    stTargetAssertion := i_stRequestedAssertion;
    nTargetAssertionID := i_nRequestedAssertionID;
	
	LogActions('New target set');
	
    xNewBP := TRUE;
    
ELSE
    IF NOT F_ValidReqID(i_nRequestedAssertionID) THEN
        
        nErrID := PMPS_CODES.BadTargetID;
    ELSIF NOT F_ValidReqID(i_TransitionAssertionID) THEN
        nErrID := PMPS_CODES.BadTransID;
	END_IF
    LogActions('Error in set new target');
    bError := TRUE;
END_IF
END_ACTION

ACTION WaitingForFinalAssertion_DO:
//Final Assertion Verification

xFinalBPInArb := fbArbiter.CheckRequest( i_nRequestedAssertionID);;
END_ACTION

ACTION WaitingForFinalAssertion_EXIT:
//Set this bool false so we can get a rising edge on the next try
xFinalBP := FALSE;
END_ACTION

ACTION WaitingForTransitionAssertion_DO:
//Transition Assertion Verification
xTranBP    := F_SafeBPCompare0Rate(stCurrentBeamParameters, i_stTransitionAssertion) AND
    fbArbiter.CheckRequest(i_TransitionAssertionID);
END_ACTION

ACTION WaitingForTransitionAssertion_EXIT:
xTranBP := FALSE;
END_ACTION

END_FUNCTION_BLOCK

// MajorComponents/InterPlcComm/FB_ArbiterToSubSys_IO
(* Exchanges preemption requests and current beam state with subsystems in arbiter
network.

2019-12-2, A. Wallace

Use in conjunction with FB_SubSysToArbiter_IO.

This FB runs in the beamline arbiter PLC (BAP). There should be one of these for every
subsystem interfaced to the BAP. Each subsystem PLC should run a sibling FB_SubSysToArbiter_IO FB.

This FB and its subordinate communicate through the ethercat connection between the subsystem PLC and the BAP.

A beam parameter set request is sent from the subsystem to this PLC, and includes a cohort number.

This cohort number (i_RequestedBP.nCohortInt) is compared to a local cohort number (nRequestedCohort). 
A request from the subsystem to update or modify its current request is indicated by an increase in the
i_RequestedBP.nCohortInt value. Then this function block updates the local arbiter request for the subsystem
and awaits confirmation. Once the new request is confirmed in the preemptive system this function block increments
the ActiveCohort value to match the nRequestedCohort. ActiveCohort is also relayed back to the subsystem
as the active cohort value in the o_CurrentBP set. The subsystem then knows its request has been heard,
and can carry out its own acknowledgement to its various requestors.

Things to note:
If a subsystem has any new or changed preemptive requests you should see the cohort value increment a bit.
If the cohort number is incrementing out of control, it usually means the subsysetm has some preemptive
request loop (two arbiters elevating to each other), or there is a RequestAdd, RequestRemove loop.

*)
FUNCTION_BLOCK FB_ArbiterToSubSys_IO
VAR_INPUT
	RequestingSystemID	:	DWORD := PMPS_GVL.EXCLUDED_ASSERTION_ID; // System ID for making requests to the supreme arbiter
    sName : STRING := 'ArbiterToSubSys';
    Reset : BOOL;
END_VAR
VAR_OUTPUT
END_VAR
VAR_IN_OUT
	Arbiter	: FB_Arbiter;
    fbFFHWO : FB_HardwareFFOutput;
END_VAR
VAR
    
	i_RequestedBP AT %I*	:	ST_BeamParams_IO; // Requested BP from subsystem
    {attribute 'pytmc' := '
        pv: RequestedBP:FromSubSys
    '}
    RequestedBP: ST_BeamParams;
    
	o_CurrentBP AT %Q* : ST_BeamParams_IO; // Current BP set
    
    // EL6692 Diagnostics
    i_Connected AT %I* : BOOL; // SYNC Inputs^External device not connected !!! Doesn't really work.
    {attribute 'pytmc' := 'pv: WcState
        io: i
        field: DESC Working counter state.
        field: ZNAM OK
        field: ONAM Error'}
    i_WcState AT %I* : BOOL := TRUE; // WcState^WcState
    {attribute 'pytmc' := 'pv: TxPDO_state
        io: i
        field: DESC PDO Transmission is OK
        field: ZNAM OK
        field: ONAM Error'}
    i_TxPDOState AT %I* : BOOL := TRUE; // SYNC Inputs^TxPDO state
    {attribute 'pytmc' := 'pv: TxPDO_toggle
        io: i
        field: DESC PDO Transmission is OK
        field: ZNAM OK
        field: ONAM Error'}
    i_TxPDOToggle AT %I* : BOOL; // TxPDO toggle
    
    // Fast faults
    ffPMPSIO_Disconnect : FB_FastFault := (i_Desc:='Issue w/ arbiter interface to subsystem, verify subsystem is OK, or ethercat connection.'); // Fast fault for ethercat issues
    nActiveCohort : UDINT := 0; // Active cohort. Updated to the req. number from the sub system after request is confirmed.
    nRequestedCohort : UDINT := 0;
    rtToggle : R_TRIG;

	
END_VAR


// Incoming request from subsystem PLC
RequestedBP := IO_TO_BP(i_RequestedBP);

// Update Arbiter with our request
rtToggle(CLK:= i_RequestedBP.xValid); // If interface resumes, reset/catch up
// xValid will go false if the PLC program on the other side is stopped. Ironically the ethercat interface continues happily.
// If subsystem cohort has incremented, update beam parameter request with our arbiter
IF rtToggle.Q THEN
    nActiveCohort := 0;    
END_IF

IF i_RequestedBP.nCohortInt > nRequestedCohort OR rtToggle.Q THEN 
    Arbiter.RemoveRequest(RequestingSystemID);
    Arbiter.AddRequest(RequestingSystemID, RequestedBP,sName);
    nRequestedCohort := i_RequestedBP.nCohortInt;    
END_IF


// Check if latest request is acknowledged by this arbiter
// Acknowledgement happens after an arbitration cycle, which means if RequestedCohort just incremented
// due to a new request, CheckRequest will be false.
IF Arbiter.CheckRequest(RequestingSystemID) THEN
    nActiveCohort := nRequestedCohort; // If it is, then the active cohort is set to the requested cohort number.
END_IF

// Sending current beam parameter set to subsystems 
o_CurrentBP := BP_TO_IO(PMPS_GVL.stCurrentBeamParameters);
o_CurrentBP.nCohortInt := nActiveCohort;


//////////////////////////////////////
// Verifying the ethercat interface health
/////////////////////////////////////
// Both of these values should be 0 for a fully valid exchange
ffPMPSIO_Disconnect.i_xOK := NOT i_WcState AND NOT i_TxPDOState;

ffPMPSIO_Disconnect(
    io_fbFFHWO := fbFFHWO,
    i_xReset := Reset,
    i_DevName := sName,
    i_TypeCode:=5);

END_FUNCTION_BLOCK

// MajorComponents/InterPlcComm/FB_SubSysToArbiter_IO
// Use on a subsystem PLC to request from the arbiter
// Run at the top of your cycle to receive the latest BP
FUNCTION_BLOCK FB_SubSysToArbiter_IO IMPLEMENTS I_HigherAuthority
VAR_INPUT
    Reset : BOOL; // Fast fault reset
    sName : STRING := 'SubSysToArbiter';
    i_bVeto : BOOL;
END_VAR
VAR_OUTPUT
END_VAR
VAR_IN_OUT
	Arbiter	: FB_Arbiter;
    fbFFHWO : FB_HardwareFFOutput;
END_VAR
VAR
    {attribute 'TcLinkTo' := 'TIIB[PMPS_PRE]^IO Inputs^CurrentBP'}
    i_stCurrentBP    AT %I* :    ST_BeamParams_IO;
    {attribute 'TcLinkTo' := 'TIIB[PMPS_PRE]^IO Outputs^RequestedBP'}
    q_stRequestedBP AT %Q* :    ST_BeamParams_IO;
    {attribute 'pytmc' := 'pv: TxPDO_toggle
        io: i'}
    {attribute 'TcLinkTo' := 'TIIB[PMPS_PRE]^SYNC Inputs^TxPDO toggle'}
    xTxPDO_toggle    AT     %I* :    BIT;
    {attribute 'pytmc' := 'pv: TxPDO_state
        io: i'}
    {attribute 'TcLinkTo' := 'TIIB[PMPS_PRE]^SYNC Inputs^TxPDO state'}
    xTxPDO_state    AT    %I*    :    BIT;
    
    
    // Fast faults
    ffPMPSIO_Disconnect : FB_FastFault := (i_Desc:='Arbiter network interface disconnected or not OP',i_DevName := sName);
    
    // A request is not considered included until the active cohort number is >= the request cohort number.
    {attribute 'pytmc' := 'pv: RequestCohort
        io: i'}
    nRequestCohort : UDINT := 0; // Request cohort
    {attribute 'pytmc' := 'pv: ActiveCohort
        io: i'}
    nActiveCohort : UDINT := 0; // Active cohort, updated by incoming BP from arbiter PLC, in the ElevateRequest arbiter call
    
    fbVetoArb : FB_VetoArbiter;

	fbLog : FB_LogMessage;
END_VAR

//Receiving current BP state
PMPS_GVL.stCurrentBeamParameters := IO_TO_BP(i_stCurrentBP);
PMPS_GVL.stCurrentBeamParameters.xValidToggle := xTxPDO_toggle; // This line must follow the one above. Sequence is important.

// Forwarding BP request for the subsystem
fbVetoArb.bVeto := i_bVeto;
fbVetoArb(HigherAuthority:=THIS^, LowerAuthority:=Arbiter, FFO:=fbFFHWO);

//Broadcasting current request
PMPS_GVL.stRequestedBeamParameters := IO_TO_BP(q_stRequestedBP);


q_stRequestedBP.xValid := TRUE; // This is set and held true here every cycle to prove the PLC on this side is still running

ffPMPSIO_Disconnect(
    i_xOK := xTxPDO_state = 0,
    io_fbFFHWO := fbFFHWO,
    i_xReset := Reset,
    i_DevName := sName,
    i_TypeCode := 6,
    i_xVetoable := FALSE
    );

METHOD CheckRequest : BOOL
VAR_INPUT
	nReqID	: DWORD;
END_VAR
VAR_INST
    xFirstTime : BOOL := TRUE;
    nId : DWORD;
END_VAR
// Check this id matches what we've seen before
IF xFirstTime THEN
    nId := nReqId;
ELSIF nId <> nReqId THEN
    fbLog(sMsg := 'SubSysToArbiter Check mismatched with a different ID', eSevr := TcEventSeverity.Error);
    RETURN;
END_IF

nActiveCohort := ULINT_TO_UDINT(i_stCurrentBP.nCohortInt);

// i_stCurrentBP.nCohortInt is incremented by the FB_ArbiterToSubSys block on the other side of the EL669* interface
CheckRequest := nRequestCohort <= nActiveCohort;
END_METHOD

METHOD RemoveRequest : BOOL
VAR_INPUT
	nReqID    :    DWORD; //StateID to remove
END_VAR
// Update internal BP request struct
q_stRequestedBP := BP_TO_IO(PMPS_GVL.cstFullBeam);

nRequestCohort := nRequestCohort + 1;

// Mark the current cohort id
q_stRequestedBP.nCohortInt := nRequestCohort;

RemoveRequest := TRUE;
END_METHOD

METHOD RequestBP : BOOL
VAR_INPUT
	(*StateID of state requesting beam parameter set*)
	nReqID	: DWORD;
	(*Requested beam params*)
	stReqBP	: ST_BeamParams;
END_VAR
// Check the request is coming from the same source we're used to

// Update internal BP request struct
q_stRequestedBP := BP_TO_IO(stReqBP);

nRequestCohort := nRequestCohort + 1;

// Mark the current cohort id
q_stRequestedBP.nCohortInt := nRequestCohort;

RequestBP := TRUE;
END_METHOD

END_FUNCTION_BLOCK

// MajorComponents/PhotonEnergyInterface/F_CalculatePhotonEnergy
FUNCTION F_CalculatePhotonEnergy : LREAL
VAR_INPUT
    (* Electron energy in GeV *)
    fElectronEnergy_GeV : LREAL;
    (* Undulator period in mm *)
    fUndulatorPeriod_mm : LREAL;
    (* Unitless undulator K parameter / strength *)
    fUndulatorStrength : LREAL;
END_VAR

VAR
    fDenominator: LREAL;
END_VAR

VAR CONSTANT
    (* GeV [electron rest mass/energy] *)
    m_e : LREAL := 0.0005109989461;
    (* Js [Planck's constant] *)
    h 	: LREAL := 6.62607004E-34;
    (* C [electron charge] *)
    e 	: LREAL := 1.6021766208E-19;
    (* m/s, speed of light *)
    c 	: LREAL := 299792458;

END_VAR

(*

Reference Python implementation

def calculate_photon_energy(electron_energy, period, k):
    '''
    Calculate photon energy, in eV.

    Parameters
    ----------
    electron_energy : float
        Electron energy in GeV

    period : float
        Undulator period, in mm

    k : float
        Undulator K parameter (strength), unitless
    '''
    m_e = 0.0005109989461  # GeV [electron rest mass/energy]
    h = 6.62607004e-34  # Js [Planck's constant]
    e = 1.6021766208e-19  # C [electron charge]
    c = 299792458  # m/s, speed of light
    return ((2. * (electron_energy / m_e) ** 2 * h * c) /
            (e * period * 1e-3 * (1 + k ** 2 / 2.)))

*)
fDenominator := (e * fUndulatorPeriod_mm * 1E-3 * (1.0 + EXPT(fUndulatorStrength, 2.0) / 2.0));
F_CalculatePhotonEnergy := (2.0 * EXPT(fElectronEnergy_GeV / m_e, 2.0) * h * c) / MAX(fDenominator, 4.94065645841247E-324);

END_FUNCTION

// MajorComponents/PhotonEnergyInterface/FB_AcceleratorLinks
FUNCTION_BLOCK FB_AcceleratorLinks
VAR_INPUT

END_VAR

VAR_OUTPUT
END_VAR


VAR

    {attribute 'pytmc' := '
        pv: eEnrg:Hgvpu
        link: BEND:DMPH:400:BACT
        field: EGU GeV
    '}
    fbHgvpuElectronEnergy : FB_LREALFromEPICS;

    {attribute 'pytmc' := '
        pv: eEnrg:SXU
        link: BEND:DMPS:400:BACT
        field: EGU GeV
    '}
    fbSxuElectronEnergy : FB_LREALFromEPICS;

END_VAR

fbHgvpuElectronEnergy();
fbSxuElectronEnergy();

END_FUNCTION_BLOCK

// MajorComponents/PhotonEnergyInterface/FB_Hgvpu
FUNCTION_BLOCK FB_Hgvpu IMPLEMENTS I_UndulatorComplex
VAR_INPUT
    fbElectronEnergy : REFERENCE TO FB_LREALFromEPICS;
END_VAR

VAR_OUTPUT
	{attribute 'pytmc' := '
        pv: CurrentPhotonEnergy
		io: i
        field: DESC Calculated current photon energy
        field: PREC 3
        field: EGU eV
    '}
	fCurrentPhotonEnergy : LREAL;
	{attribute 'pytmc' := '
        pv: TargetPhotonEnergy
		io: i
        field: DESC Calculated desired photon energy
        field: PREC 3
        field: EGU eV
    '}
	fTargetPhotonEnergy : LREAL;
    {attribute 'pytmc' := '
        pv: SeedUndulatorNumber
		io: i
        field: DESC Seed undulator number
    '}
	nSeedUndulator : UDINT; // Set to zero when no undulators are active
    {attribute 'pytmc' := '
        pv: TargetSeedUndulatorNumber
		io: i
        field: DESC Seed undulator number for target K
    '}
	nTargetSeedUndulator : UDINT; // Set to zero when no undulators are active
END_VAR


VAR
    // From lcls-srv01: grep -e KDes  /u1/lcls/epics/ioc/data/ioc-undh-uc*/iocInfo/IOC.pvlist |sort

    {attribute 'pytmc' := 'pv: 24; link: 2450:'}
    fbSegment_24 : FB_UndulatorSegment;

    {attribute 'pytmc' := 'pv: 25; link: 2550:'}
    fbSegment_25 : FB_UndulatorSegment;

    {attribute 'pytmc' := 'pv: 26; link: 2650:'}
    fbSegment_26 : FB_UndulatorSegment;

    {attribute 'pytmc' := 'pv: 27; link: 2750:'}
    fbSegment_27 : FB_UndulatorSegment;

    {attribute 'pytmc' := 'pv: 29; link: 2950:'}
    fbSegment_29 : FB_UndulatorSegment;

    {attribute 'pytmc' := 'pv: 30; link: 3050:'}
    fbSegment_30 : FB_UndulatorSegment;

    {attribute 'pytmc' := 'pv: 31; link: 3150:'}
    fbSegment_31 : FB_UndulatorSegment;

    {attribute 'pytmc' := 'pv: 32; link: 3250:'}
    fbSegment_32 : FB_UndulatorSegment;

    {attribute 'pytmc' := 'pv: 33; link: 3350:'}
    fbSegment_33 : FB_UndulatorSegment;

    {attribute 'pytmc' := 'pv: 34; link: 3450:'}
    fbSegment_34 : FB_UndulatorSegment;

    {attribute 'pytmc' := 'pv: 35; link: 3550:'}
    fbSegment_35 : FB_UndulatorSegment;

    {attribute 'pytmc' := 'pv: 36; link: 3650:'}
    fbSegment_36 : FB_UndulatorSegment;

    {attribute 'pytmc' := 'pv: 37; link: 3750:'}
    fbSegment_37 : FB_UndulatorSegment;

    {attribute 'pytmc' := 'pv: 38; link: 3850:'}
    fbSegment_38 : FB_UndulatorSegment;

    {attribute 'pytmc' := 'pv: 39; link: 3950:'}
    fbSegment_39 : FB_UndulatorSegment;

    {attribute 'pytmc' := 'pv: 40; link: 4050:'}
    fbSegment_40 : FB_UndulatorSegment;

    {attribute 'pytmc' := 'pv: 41; link: 4150:'}
    fbSegment_41 : FB_UndulatorSegment;

    {attribute 'pytmc' := 'pv: 42; link: 4250:'}
    fbSegment_42 : FB_UndulatorSegment;

    {attribute 'pytmc' := 'pv: 43; link: 4350:'}
    fbSegment_43 : FB_UndulatorSegment;

    {attribute 'pytmc' := 'pv: 44; link: 4450:'}
    fbSegment_44 : FB_UndulatorSegment;

    {attribute 'pytmc' := 'pv: 45; link: 4550:'}
    fbSegment_45 : FB_UndulatorSegment;

    {attribute 'pytmc' := 'pv: 46; link: 4650:'}
    fbSegment_46 : FB_UndulatorSegment;

    fbSegment : ARRAY [iLowBound_LUnd..iHighBound_LUnd] OF POINTER TO FB_UndulatorSegment;
    fbCurrentSegment : REFERENCE TO FB_UndulatorSegment;

    iIndex : UDINT;

    bInitialized : BOOL := FALSE;

END_VAR

VAR CONSTANT
    {attribute 'pytmc' := '
		pv: FirstSegment
		io: i
	'}
    iLowBound_LUnd  : UDINT := 24;
	
    {attribute 'pytmc' := '
		pv: LastSegment
		io: i
	'}
    iHighBound_LUnd : UDINT := 46;
	
    {attribute 'pytmc' := '
        pv: Period
        io: i
        field: EGU mm
    '}
    fPeriod_mm_LUnd : LREAL := 26.0;
	
	{attribute 'pytmc' := '
        pv: LowK
        io: i
    '}
	fLowK_LUnd : LREAL := 0.54;
	
	{attribute 'pytmc' := '
        pv: HiK
        io: i
    '}
	fHiK_LUnd : LREAL := 2.6;
END_VAR

IF NOT bInitialized THEN
	Init();
END_IF

UndAdrUpdate();

nSeedUndulator := 0;
nTargetSeedUndulator := 0;

FOR iIndex := iLowBound_LUnd TO iHighBound_LUnd DO
    IF fbSegment[iIndex] <> 0 THEN
        fbCurrentSegment REF= fbSegment[iIndex]^;
        fbCurrentSegment(fbElectronEnergy:=fbElectronEnergy);
		
		//Mark the seed undulator, first undulator operating within K bounds
		IF fbCurrentSegment.xActive AND nSeedUndulator = 0 THEN
			nSeedUndulator := iIndex;
			fCurrentPhotonEnergy := fbCurrentSegment.fPhotonEnergyAct;
		END_IF
        
        IF fbCurrentSegment.xTargetActive AND nTargetSeedUndulator = 0 THEN
			nTargetSeedUndulator := iIndex;
			fTargetPhotonEnergy := fbCurrentSegment.fPhotonEnergyDes;
		END_IF
    END_IF
END_FOR

IF nSeedUndulator = 0 THEN
	fCurrentPhotonEnergy := 0;
END_IF

IF nTargetSeedUndulator = 0 THEN
    fTargetPhotonEnergy := 0;
END_IF

ACTION Init:

UndAdrUpdate();


    FOR iIndex := iLowBound_LUnd TO iHighBound_LUnd DO
            IF fbSegment[iIndex] <> 0 THEN
            fbCurrentSegment REF= fbSegment[iIndex]^;
            fbCurrentSegment.fPeriod_mm := fPeriod_mm_LUnd;
			fbCurrentSegment.fLowK := fLowK_LUnd;
			fbCurrentSegment.fHiK := fHiK_LUnd;
        END_IF
    END_FOR

    bInitialized := TRUE;
END_ACTION

PROPERTY rCurrentPhotonEnergy : REAL
GET
rCurrentPhotonEnergy := fCurrentPhotonEnergy;
END_GET
END_PROPERTY

PROPERTY rTargetPhotonEnergy : REAL
GET
rTargetPhotonEnergy := fTargetPhotonEnergy;
END_GET
END_PROPERTY

ACTION UndAdrUpdate:
fbSegment[24] := ADR(fbSegment_24);
fbSegment[25] := ADR(fbSegment_25);
fbSegment[26] := ADR(fbSegment_26);
fbSegment[27] := ADR(fbSegment_27);
fbSegment[28] := 0;
fbSegment[29] := ADR(fbSegment_29);
fbSegment[30] := ADR(fbSegment_30);
fbSegment[31] := ADR(fbSegment_31);
fbSegment[32] := ADR(fbSegment_32);
fbSegment[33] := ADR(fbSegment_33);
fbSegment[34] := ADR(fbSegment_34);
fbSegment[35] := ADR(fbSegment_35);
fbSegment[36] := ADR(fbSegment_36);
fbSegment[37] := ADR(fbSegment_37);
fbSegment[38] := ADR(fbSegment_38);
fbSegment[39] := ADR(fbSegment_39);
fbSegment[40] := ADR(fbSegment_40);
fbSegment[41] := ADR(fbSegment_41);
fbSegment[42] := ADR(fbSegment_42);
fbSegment[43] := ADR(fbSegment_43);
fbSegment[44] := ADR(fbSegment_44);
fbSegment[45] := ADR(fbSegment_45);
fbSegment[46] := ADR(fbSegment_46);
END_ACTION

END_FUNCTION_BLOCK

// MajorComponents/I_UndulatorComplex
INTERFACE I_UndulatorComplex

PROPERTY rCurrentPhotonEnergy : REAL
GET
END_GET
END_PROPERTY

PROPERTY rTargetPhotonEnergy : REAL
GET
END_GET
END_PROPERTY

END_INTERFACE

// MajorComponents/PhotonEnergyInterface/FB_UndulatorSegment
FUNCTION_BLOCK FB_UndulatorSegment
VAR_INPUT
    (* Undulator period in millimeters, to be set by subclasses *)
    fPeriod_mm : LREAL := 1.0;
    fbElectronEnergy : REFERENCE TO FB_LREALFromEPICS;
	
	fLowK : LREAL := 0;
	fHiK : LREAL := 6;
	fKRangeHyst : LREAL := 0.01;
END_VAR

VAR_OUTPUT
    {attribute 'pytmc' := '
        pv: eVAct
        field: DESC Calculated photon energy
        field: PREC 3
        field: EGU eV
    '}
    fPhotonEnergyAct : LREAL;

    {attribute 'pytmc' := '
        pv: eVDes
        field: DESC Calculated desired photon energy
        field: PREC 3
        field: EGU eV
    '}
    fPhotonEnergyDes : LREAL;
	
	{attribute 'pytmc' := '
        pv: Active
		io: i
        field: DESC Undulator is considered active
    '}
	xActive : BOOL; // Undulator is considered active
    
    {attribute 'pytmc' := '
        pv: TargetActive
		io: i
        field: DESC Target K would make und active
    '}
	xTargetActive : BOOL; // Undulator is considered active at this target
    
    {attribute 'pytmc' := '
        pv: KAct
		io: i
        field: DESC Current K
    '}
    fKAct : LREAL;
    
    {attribute 'pytmc' := '
        pv: KDes
		io: i
        field: DESC Target K
    '}
    fKDes : LREAL;
    
        {attribute 'pytmc' := '
        pv: KActValid
		io: i
        field: DESC Current K Readback Valid
    '}
    bKActValid : BOOL;
    
    {attribute 'pytmc' := '
        pv: KDesValid
		io: i
        field: DESC Target K Readback Valid
    '}
    bKDesValid : BOOL;
    
END_VAR

VAR
    {attribute 'pytmc' := '
        pv: KDes
        link: KDes
    '}
    fbKDesired : FB_LREALFromEPICS;

    {attribute 'pytmc' := '
        pv: KAct
        link: KAct
    '}
    fbKActual : FB_LREALFromEPICS;

END_VAR

fbKDesired();
fbKActual();

fKAct := fbKActual.fValue;
bKActValid := fbKActual.bValid;
fKDes := fbKDesired.fValue;
bKDesValid := fbKDesired.bvalid;

IF __ISVALIDREF(fbElectronEnergy) THEN

    IF fbKActual.bValid AND fbElectronEnergy.bValid THEN
        fPhotonEnergyAct := F_CalculatePhotonEnergy(
            fElectronEnergy_GeV:=fbElectronEnergy.fValue,
            fUndulatorPeriod_mm:=fPeriod_mm,
            fUndulatorStrength:=fbKActual.fValue
        );
		
		//Set this undulator active if actual K is within operational range
		xActive S= fLowK <= fbKActual.fValue AND fbKActual.fValue <= fHiK AND
		(fbKActual.bValid AND fbKActual.bValid);
		xActive R= (fLowK - fKRangeHyst) > fbKActual.fValue OR fbKActual.fValue > (fHiK + fKRangeHyst) OR
					(NOT fbKActual.bValid OR NOT fbKActual.bValid);
                    
        //Set this undulator active if target K is within operational range
		xTargetActive S= fLowK <= fbKDesired.fValue AND fbKDesired.fValue <= fHiK AND
		(fbKDesired.bValid AND fbKDesired.bValid);
		xTargetActive R= (fLowK - fKRangeHyst) > fbKDesired.fValue OR fbKDesired.fValue > (fHiK + fKRangeHyst) OR
					(NOT fbKDesired.bValid OR NOT fbKDesired.bValid);
    END_IF

    IF fbKDesired.bValid AND fbElectronEnergy.bValid THEN
        fPhotonEnergyDes := F_CalculatePhotonEnergy(
            fElectronEnergy_GeV:=fbElectronEnergy.fValue,
            fUndulatorPeriod_mm:=fPeriod_mm,
            fUndulatorStrength:=fbKDesired.fValue
        );
    END_IF

END_IF

END_FUNCTION_BLOCK

// MajorComponents/PhotonEnergyInterface/FB_KPhotonEnergy
FUNCTION_BLOCK FB_KPhotonEnergy EXTENDS FB_PhotonEnergy
VAR_INPUT
END_VAR
VAR_OUTPUT
END_VAR
VAR
    {attribute 'pytmc' := '
        pv: eEnrg
        link: BEND:DMPS:400:BACT
        field: EGU GeV
    '}
    fbSxuElectronEnergy : FB_LREALFromEPICS;
    
    {attribute 'pytmc' := '
        pv: EEnergy
		io: i
        field: DESC Electron Energy
        field: EGU GeV
    '}
    fElectronEnergyVal : LREAL;
    
    {attribute 'pytmc' := '
        pv: EEnergyValid
		io: i
        field: DESC Electron Energy Valid
    '}
    bElectronEnergyValid : BOOL;
	
    {attribute 'pytmc' := '
        pv: UND
        link: USEG:UNDS:
    '}
    fbSxu : FB_SXU;

END_VAR

// Update PVs
fbSxuElectronEnergy();

fElectronEnergyVal := fbSxuElectronEnergy.fValue;
bElectronEnergyValid := fbSxuElectronEnergy.bValid;

fbSxu(fbElectronEnergy:=fbSxuElectronEnergy);

SUPER^(BP:=SUPER^.BP, Undulator:=fbSxu );

END_FUNCTION_BLOCK

// MajorComponents/PhotonEnergyInterface/FB_PhotonEnergy
FUNCTION_BLOCK FB_PhotonEnergy
VAR_INPUT
    Undulator : I_UndulatorComplex;
END_VAR
VAR_OUTPUT
END_VAR
VAR_IN_OUT
	BP : ST_BeamParams;
END_VAR
VAR
    nCurrentPhotonEnergyBitmask : UDINT;
	nTargetPhotonEnergyBitmask : UDINT;
END_VAR


//Update BP
nCurrentPhotonEnergyBitmask := F_eVRangeCalculator(Undulator.rCurrentPhotonEnergy, nCurrentPhotonEnergyBitmask);
nTargetPhotonEnergyBitmask := F_eVRangeCalculator(Undulator.rTargetPhotonEnergy, nTargetPhotonEnergyBitmask);

BP.neVRange := nCurrentPhotonEnergyBitmask OR nTargetPhotonEnergyBitmask;

END_FUNCTION_BLOCK

// MajorComponents/PhotonEnergyInterface/FB_SXU
FUNCTION_BLOCK FB_SXU IMPLEMENTS I_UndulatorComplex
VAR_INPUT
    fbElectronEnergy : REFERENCE TO FB_LREALFromEPICS;
END_VAR

VAR_OUTPUT
    {attribute 'pytmc' := '
        pv: CurrentPhotonEnergy
		io: i
        field: DESC Calculated current photon energy
        field: PREC 3
        field: EGU eV
    '}
	fCurrentPhotonEnergy : LREAL;
	{attribute 'pytmc' := '
        pv: TargetPhotonEnergy
		io: i
        field: DESC Calculated desired photon energy
        field: PREC 3
        field: EGU eV
    '}
	fTargetPhotonEnergy : LREAL;
	    {attribute 'pytmc' := '
        pv: SeedUndulatorNumber
		io: i
        field: DESC Seed undulator number
    '}
	nSeedUndulator : UDINT; // Set to zero when no undulators are active
    {attribute 'pytmc' := '
        pv: TargetSeedUndulatorNumber
		io: i
        field: DESC Seed undulator number for target K
    '}
	nTargetSeedUndulator : UDINT; // Set to zero when no undulators are active
END_VAR



VAR
    // From lcls-srv01: grep -e KDes  /u1/lcls/epics/ioc/data/sioc-unds-uc*/iocInfo/IOC.pvlist |sort


    {attribute 'pytmc' := 'pv: 26; link: 2650:'}
    fbSegment_26 : FB_UndulatorSegment;

    {attribute 'pytmc' := 'pv: 27; link: 2750:'}
    fbSegment_27 : FB_UndulatorSegment;

    {attribute 'pytmc' := 'pv: 28; link: 2850:'}
    fbSegment_28 : FB_UndulatorSegment;

    {attribute 'pytmc' := 'pv: 29; link: 2950:'}
    fbSegment_29 : FB_UndulatorSegment;

    {attribute 'pytmc' := 'pv: 30; link: 3050:'}
    fbSegment_30 : FB_UndulatorSegment;

    {attribute 'pytmc' := 'pv: 31; link: 3150:'}
    fbSegment_31 : FB_UndulatorSegment;

    {attribute 'pytmc' := 'pv: 32; link: 3250:'}
    fbSegment_32 : FB_UndulatorSegment;

    {attribute 'pytmc' := 'pv: 33; link: 3350:'}
    fbSegment_33 : FB_UndulatorSegment;

    {attribute 'pytmc' := 'pv: 34; link: 3450:'}
    fbSegment_34 : FB_UndulatorSegment;

    {attribute 'pytmc' := 'pv: 36; link: 3650:'}
    fbSegment_36 : FB_UndulatorSegment;

    {attribute 'pytmc' := 'pv: 37; link: 3750:'}
    fbSegment_37 : FB_UndulatorSegment;

    {attribute 'pytmc' := 'pv: 38; link: 3850:'}
    fbSegment_38 : FB_UndulatorSegment;

    {attribute 'pytmc' := 'pv: 39; link: 3950:'}
    fbSegment_39 : FB_UndulatorSegment;

    {attribute 'pytmc' := 'pv: 40; link: 4050:'}
    fbSegment_40 : FB_UndulatorSegment;

    {attribute 'pytmc' := 'pv: 41; link: 4150:'}
    fbSegment_41 : FB_UndulatorSegment;

    {attribute 'pytmc' := 'pv: 42; link: 4250:'}
    fbSegment_42 : FB_UndulatorSegment;

    {attribute 'pytmc' := 'pv: 43; link: 4350:'}
    fbSegment_43 : FB_UndulatorSegment;

    {attribute 'pytmc' := 'pv: 44; link: 4450:'}
    fbSegment_44 : FB_UndulatorSegment;

    {attribute 'pytmc' := 'pv: 45; link: 4550:'}
    fbSegment_45 : FB_UndulatorSegment;

    {attribute 'pytmc' := 'pv: 46; link: 4650:'}
    fbSegment_46 : FB_UndulatorSegment;

    {attribute 'pytmc' := 'pv: 47; link: 4750:'}
    fbSegment_47 : FB_UndulatorSegment;



    fbSegment : ARRAY [iLowBound..iHighBound] OF POINTER TO FB_UndulatorSegment;
    fbCurrentSegment : REFERENCE TO FB_UndulatorSegment;

    iIndex : UDINT;

    bInitialized : BOOL := FALSE;

END_VAR

VAR CONSTANT
    {attribute 'pytmc' := '
		pv: FirstSegment
		io: i'}
    iLowBound  : UDINT := 26;
    {attribute 'pytmc' := '
		pv: LastSegment
	 	io: i'}
    iHighBound : UDINT := 47;
    {attribute 'pytmc' := '
        pv: Period
        io: i
        field: EGU mm
    '}
    fPeriod_mm : LREAL := 39.0;
    {attribute 'pytmc' := '
        pv: LowK
        io: i
    '}
	fLowK : LREAL := 1.5;
	
	{attribute 'pytmc' := '
        pv: HiK
        io: i
    '}
	fHiK : LREAL := 5.7; 
END_VAR



IF NOT bInitialized THEN
    Init();
END_IF

UndAdrUpdate();

nSeedUndulator := 0;
nTargetSeedUndulator := 0;

FOR iIndex := iLowBound TO iHighBound DO
    IF fbSegment[iIndex] <> 0 THEN
        fbCurrentSegment REF= fbSegment[iIndex]^;
        fbCurrentSegment(fbElectronEnergy:=fbElectronEnergy);
		
		//Mark the seed undulator, first undulator operating within K bounds
		IF fbCurrentSegment.xActive AND nSeedUndulator = 0 THEN
			nSeedUndulator := iIndex;
			fCurrentPhotonEnergy := fbCurrentSegment.fPhotonEnergyAct;
		END_IF
        
        IF fbCurrentSegment.xTargetActive AND nTargetSeedUndulator = 0 THEN
			nTargetSeedUndulator := iIndex;
			fTargetPhotonEnergy := fbCurrentSegment.fPhotonEnergyDes;
		END_IF
    END_IF
END_FOR

IF nSeedUndulator = 0 THEN
	fCurrentPhotonEnergy := 0;
END_IF

IF nTargetSeedUndulator = 0 THEN
    fTargetPhotonEnergy := 0;
END_IF

ACTION Init:

UndAdrUpdate();

FOR iIndex := iLowBound TO iHighBound DO
        IF fbSegment[iIndex] <> 0 THEN
        fbCurrentSegment REF= fbSegment[iIndex]^;
		fbCurrentSegment.fPeriod_mm := fPeriod_mm;
		fbCurrentSegment.fLowK := fLowK;
		fbCurrentSegment.fHiK := fHiK;
    END_IF
END_FOR
bInitialized := TRUE;
END_ACTION

PROPERTY rCurrentPhotonEnergy : REAL
GET
rCurrentPhotonEnergy := fCurrentPhotonEnergy;
END_GET
END_PROPERTY

PROPERTY rTargetPhotonEnergy : REAL
GET
rTargetPhotonEnergy := fTargetPhotonEnergy;
END_GET
END_PROPERTY

ACTION UndAdrUpdate:

fbSegment[26] := ADR(fbSegment_26);
fbSegment[27] := ADR(fbSegment_27);
fbSegment[28] := ADR(fbSegment_28);
fbSegment[29] := ADR(fbSegment_29);
fbSegment[30] := ADR(fbSegment_30);
fbSegment[31] := ADR(fbSegment_31);
fbSegment[32] := ADR(fbSegment_32);
fbSegment[33] := ADR(fbSegment_33);
fbSegment[34] := ADR(fbSegment_34);
fbSegment[35] := 0;
fbSegment[36] := ADR(fbSegment_36);
fbSegment[37] := ADR(fbSegment_37);
fbSegment[38] := ADR(fbSegment_38);
fbSegment[39] := ADR(fbSegment_39);
fbSegment[40] := ADR(fbSegment_40);
fbSegment[41] := ADR(fbSegment_41);
fbSegment[42] := ADR(fbSegment_42);
fbSegment[43] := ADR(fbSegment_43);
fbSegment[44] := ADR(fbSegment_44);
fbSegment[45] := ADR(fbSegment_45);
fbSegment[46] := ADR(fbSegment_46);
fbSegment[47] := ADR(fbSegment_47);
END_ACTION

END_FUNCTION_BLOCK

// MajorComponents/PhotonEnergyInterface/FB_LPhotonEnergy
FUNCTION_BLOCK FB_LPhotonEnergy EXTENDS FB_PhotonEnergy
VAR_INPUT
END_VAR
VAR_OUTPUT
END_VAR
VAR
	{attribute 'pytmc' := '
        pv: eEnrg
        link: BEND:DMPH:400:BACT
        field: EGU GeV
    '}
    fbHgvpuElectronEnergy : FB_LREALFromEPICS;
	
    {attribute 'pytmc' := '
        pv: EEnergy
		io: i
        field: DESC Electron Energy
        field: EGU GeV
    '}
    fElectronEnergyVal : LREAL;
    
    {attribute 'pytmc' := '
        pv: EEnergyValid
		io: i
        field: DESC Electron Energy Valid
    '}
    bElectronEnergyValid : BOOL;
    
	{attribute 'pytmc' := '
        pv: UND
        link: USEG:UNDH:
    '}
    fbHgvpu : FB_Hgvpu;
	
END_VAR

// Update PVs
fbHgvpuElectronEnergy();

fElectronEnergyVal := fbHgvpuElectronEnergy.fValue;
bElectronEnergyValid := fbHgvpuElectronEnergy.bValid;

fbHgvpu(fbElectronEnergy:=fbHgvpuElectronEnergy);

SUPER^(BP:=SUPER^.BP, Undulator:=fbHgvpu );

END_FUNCTION_BLOCK

// MajorComponents/PMPS_MPS_Interface/FB_BeamClassOutputs
(*
Sets the beam class assertion lines for a given beam class.
*)
FUNCTION_BLOCK FB_BeamClassOutputs
VAR_INPUT
    BP : ST_BeamParams;
END_VAR
VAR_OUTPUT
END_VAR
VAR
    nBeamClass   :    BYTE;
    wBeamClass    :    BYTE;

    InitCounter: BYTE;
    counter    :    INT;
    
    // Beam class lines are restricted to 8 channels in the current design, since
    // there are no plans to use all 16. Channels 1-7 may be allocated to any other
    // beam classes so long as they are ordered least to greatest.
    // Channel 8 is reserved for full beam.
    {attribute 'pytmc' := 'pv: BeamClassChannel
        io: i
        field: DESC Hardwire channel state'}
        epicsBitmap : WORD;
        
    {attribute 'TcLinkTo' := '[1] := TIIB[PMPS_Premp]^Channel 1^Output;
                              [2] := TIIB[PMPS_Premp]^Channel 2^Output;
                              [3] := TIIB[PMPS_Premp]^Channel 3^Output;
                              [4] := TIIB[PMPS_Premp]^Channel 4^Output;
                              
                              [5] := TIIB[PMPS_Premp]^Channel 5^Output;
                              [6] := TIIB[PMPS_Premp]^Channel 6^Output;
                              [7] := TIIB[PMPS_Premp]^Channel 7^Output;
                              [8] := TIIB[PMPS_Premp]^Channel 8^Output;'} // 8 - Full beam
    q_BC_ASSERTION_LINES    AT    %Q*    : ARRAY [1..MAX_BEAM_CLASS_LINES] OF    BOOL;
END_VAR
VAR CONSTANT
    MAX_BEAM_CLASS_LINES : BYTE := 8;
    BC_1HZ : BYTE := 1;
    BC_10HZ : BYTE := 2;
    BC_FULL : BYTE := 16;
END_VAR


// Determine BC
IF BP.nRate >= 120 THEN
    nBeamClass := BC_FULL;
ELSIF BP.nRate >= 10 THEN
    nBeamClass := BC_10HZ;
ELSIF BP.nRate >= 1 THEN
    nBeamClass := BC_1HZ;
ELSE
	nBeamClass := 0;
END_IF


//Assert Beam Class
////////////////////////////////////
//0x0 = 0000 0000 0000 0000
//0x1 = 0000 0000 0000 0001
//0xF = 1111 1111 1111 1111

//Initialize BC lines to zero on every pass
FOR InitCounter := 1 TO MAX_BEAM_CLASS_LINES DO
    q_BC_ASSERTION_LINES[InitCounter] := FALSE;
END_FOR

//Set BC lines according to beam class
//A BC of 0x0 would pass over this loop, setting none of the lines high
// , as FOR loops check the initialized variable at the top to see if it's >
// than the "TO" variable.
FOR wBeamClass:=1 TO MIN(MAX_BEAM_CLASS_LINES-1, nBeamClass) DO
    q_BC_ASSERTION_LINES[wBeamClass] := TRUE;
END_FOR

q_BC_ASSERTION_LINES[8] := nBeamClass = 16; //Set channel 8 true if BC is 16


// Readbacks for EPICS
epicsBitmap.0 := q_BC_ASSERTION_LINES[1];
epicsBitmap.1 := q_BC_ASSERTION_LINES[2];
epicsBitmap.2 := q_BC_ASSERTION_LINES[3];
epicsBitmap.3 := q_BC_ASSERTION_LINES[4];

epicsBitmap.4 := q_BC_ASSERTION_LINES[5];
epicsBitmap.5 := q_BC_ASSERTION_LINES[6];
epicsBitmap.6 := q_BC_ASSERTION_LINES[7];
epicsBitmap.7 := q_BC_ASSERTION_LINES[8];

END_FUNCTION_BLOCK

// MajorComponents/PMPS_MPS_Interface/FB_CTLS_Outputs
(*
Controls auxiliary beam class outputs.

1-3 are mapped to control the Cu beamline rate via the LCLS II MPS.

Maps beam rate requests to 1, 10, or full rate beam for Cu linac.

*)
FUNCTION_BLOCK FB_CTLS_Outputs
VAR_INPUT
    BP    :    ST_BeamParams;
END_VAR
VAR_OUTPUT
END_VAR
VAR
    {attribute 'pytmc' := 'pv: CTLSChannel
        io: i
        field: DESC CTLS Rate Control hardwire channel state'}
    epicsBitmap : WORD;
        
    {attribute 'TcLinkTo' := '[1] := TIIB[PMPS_Premp]^Channel 9^Output;
                              [2] := TIIB[PMPS_Premp]^Channel 10^Output;
                              [3] := TIIB[PMPS_Premp]^Channel 11^Output;'}
    q_CLTS_ASSERTION_LINES    AT    %Q*    : ARRAY [1..3] OF    BOOL;  
    
    
    
END_VAR


// CLTS 1Hz
q_CLTS_ASSERTION_LINES[1] := BP.nRate >= 1;
// CLTS 10Hz
q_CLTS_ASSERTION_LINES[2] := BP.nRate >= 10;
// CLTS Full rate
q_CLTS_ASSERTION_LINES[3] := BP.nRate >= 120;


epicsBitMap.0 := q_CLTS_ASSERTION_LINES[1];
epicsBitMap.1 := q_CLTS_ASSERTION_LINES[2];
epicsBitMap.2 := q_CLTS_ASSERTION_LINES[3];

END_FUNCTION_BLOCK

// MajorComponents/PMPS_MPS_Interface/FB_PhotonEnergyWatcher
(*
A. Wallace 2019-4-22
The photon energy watcher ensures the current and target photon energy is within
the arbirated bounds. Target in this case means, the calculated target photon energy
from the PVs that control the mechatronics of the undulators/ the electron energy.

If there are control PVs that match the monitor PVs, the control PVs are used to 
calculate a "target" photon energy. This is supposed to cover when the undulators/
electron energy is transitioning.

The abritrated bounds come from a simple AND of all the permitted ranges. See
the arbitrate action of the arbiter FB.

Note, this protection logic does not account for beam-off when determining fast-fault
status. If a device is requesting a limited range of eV, this request must be honored,
regardless of current beam-rate.
*)
{attribute 'reflection'}
FUNCTION_BLOCK FB_PhotonEnergyWatcher
VAR_INPUT
    i_stCurrentBeamParams    :    ST_BeamParams; //Link to global beam params
    i_stMachineTargetBeamParams    :    ST_BeamParams; //Link to global machine target beam params
    i_stRequestedBeamParams    :    ST_BeamParams; //Link to arbiter output or beam param. requestor
    // Reset fault
    i_xReset: BOOL;
    sName : STRING := 'PhotonEnergyWatcher';
END_VAR
VAR_OUTPUT
END_VAR
VAR_IN_OUT
    io_fbFFHWO    :    FB_HardwareFFOutput;
END_VAR
VAR
    xPhotonEnergyWithinBounds    :    BOOL;
    fbFF    :    FB_FastFault :=(
        i_DevName := sName,
        i_Desc := 'Fault occurs when the calculated machine photon energy (K value calculated by undulator gap, and electron energy) falls outside the permitted range.',
        i_TypeCode := 7 );
        
   {attribute 'pytmc' := '
        pv: ResidualPhotonEnergies
		io: i
        archive: 1Hz monitor
        field: DESC Portions of beam eV not permitted
        field: EGU eV-bitmask
    '}
    evResidual : DWORD;
    
    fbLog : FB_LogMessage := (
        eSubSystem := E_Subsystem.MPS,
        eSevr := TcEventSeverity.Critical
        );
    bLogOneShot : BOOL;
    sDevName : T_MaxString := 'Photon Energy Watcher';
    
    fbGetHN : FB_GetHostName;
    bInit : BOOL := TRUE;
    
    {attribute 'instance-path'}
    {attribute 'noinit'}
    sPath    :    T_MaxString;
    
    fbStr : FB_FormatString := (
        sOut := 'Non-zero photon energy residual: %32b; Req: %32b; Act: %32b');
END_VAR

IF bInit THEN
    fbGetHN(bExecute:=TRUE);
    bInit R= NOT fbGetHN.bBusy;
END_IF
    
xPhotonEnergyWithinBounds := (i_stCurrentBeamParams.neVRange AND i_stRequestedBeamParams.neVRange) = i_stCurrentBeamParams.neVRange;

evResidual := (i_stCurrentBeamParams.neVRange XOR i_stRequestedBeamParams.neVRange) AND i_stCurrentBeamParams.neVRange;

IF evResidual <> 0 AND bLogOneShot THEN
    fbLog.sJson := F_PMPS_JSON(
        CONCAT(fbGetHN.sHostName, sDevName),
        sPath,
        PMPS_CODES.PEW_FAULT);
    
    fbStr.arg1 := F_DWORD(evResidual);
    fbStr.arg2 := F_DWORD(i_stCurrentBeamParams.neVRange);
    fbStr.arg3 := F_DWORD(i_stRequestedBeamParams.neVRange);
    
    fbStr();
        
    fbLog(sMsg:=fbStr.sOut);
    bLogOneShot := FALSE;
ELSIF evResidual = 0 THEN
    bLogOneShot := TRUE;
END_IF

fbFF(i_xOK := xPhotonEnergyWithinBounds,
    io_fbFFHWO := io_fbFFHWO,);

END_FUNCTION_BLOCK

// MajorComponents/SimulationFB/FB_eVSimulator
(* eV Simulator
A. Wallace 2019-8-30

Adds noise to the eV and changes eV position occasionally.
*)
FUNCTION_BLOCK FB_eVSimulator
VAR_INPUT
    NoiseLevel	:	REAL	:= 0; // eV Noise
    ChangeTime : TIME := T#10S;
END_VAR
VAR_OUTPUT
    eV	:	REAL := 300;
END_VAR
VAR
    eVRange : REAL := 1600;
    timer: TON;
    eVRand	:	DRAND :=(Seed:=0);
    NoiseRand : DRAND := (Seed:=0);
END_VAR


timer(in:=TRUE, PT:=ChangeTime);

//Occasionally change eV
IF timer.Q THEN
    timer(in:=FALSE);
    eVRand();
    eV := LIMIT(0, eVRange*LREAL_TO_REAL(eVRand.Num), eVRange);
END_IF

// Noise generation
NoiseRand();
eV := eV + NoiseLevel*LREAL_TO_REAL(NoiseRand.Num);
NoiseRand();
eV := LIMIT(0, ev - NoiseLevel*LREAL_TO_REAL(NoiseRand.Num), eVRange);

END_FUNCTION_BLOCK

// MajorComponents/SimulationFB/FB_MachineSimulator
(* Simulates the machine responding to requests by adding a bit of delay/ ramps
*)
FUNCTION_BLOCK FB_MachineSimulator
VAR_INPUT
    i_stAssertedParams    :    ST_BeamParams;
    i_xFault    :    BOOL;
    
    xEnableAtt : BOOL;
    xEnablePE : BOOL;
    xEnableRate : BOOL;
END_VAR
VAR_IN_OUT
    iq_stMachineParams    :    ST_BeamParams;
END_VAR
VAR
    nTargetTran: REAL;
    tonTranTimer    :    TON := (
        PT := T#2S
        );
    fTargetPP_mJ: REAL;
    tonPPETimer: TON := (
        PT := T#2S
    );
END_VAR


//Attenuation
IF xEnableAtt THEN
    IF i_stAssertedParams.nTran <> nTargetTran THEN
        tonTranTimer(IN:=FALSE);
        nTargetTran := i_stAssertedParams.nTran;
    ELSIF NOT tonTranTimer.Q THEN
        tonTranTimer(IN:=TRUE);
    ELSE
        iq_stMachineParams.nTran := nTargetTran;
    END_IF
END_IF
    
//Pulse Energy
(*
IF xEnablePE THEN
    IF i_stAssertedParams.fPP_mJ <> fTargetPP_mJ THEN
        tonPPETimer(IN:=FALSE);
        fTargetPP_mJ := i_stAssertedParams.fPP_mJ;
    ELSIF NOT tonTranTimer.Q THEN
        tonPPETimer(IN:=TRUE);
    ELSE
        iq_stMachineParams.fPP_mJ := fTargetPP_mJ;
    END_IF
END_IF
*)
//Rate
IF xEnableRate THEN
    IF i_xFault THEN
        iq_stMachineParams.nRate := 0;
    ELSE
        iq_stMachineParams.nRate := i_stAssertedParams.nRate;
    END_IF
END_IF

END_FUNCTION_BLOCK

// MajorComponents/Stoppers/FB_KStopper
FUNCTION_BLOCK FB_KStopper EXTENDS FB_StopperWatcher
VAR_INPUT
END_VAR
VAR_OUTPUT
END_VAR
VAR_IN_OUT
END_VAR
VAR
END_VAR

SUPER^(stCurrentBP:=SUPER^.stCurrentBP);

METHOD FB_init : BOOL
VAR_INPUT
    bInitRetains : BOOL; // if TRUE, the retain variables are initialized (warm start / cold start)
    bInCopyCode : BOOL;  // if TRUE, the instance afterwards gets moved into the copy code (online change)
    eStopper : K_Stopper;
    sStopperName : STRING;
END_VAR
Stopper := eStopper;
StopperName := sStopperName;
END_METHOD

END_FUNCTION_BLOCK

// MajorComponents/Stoppers/FB_StopperWatcher
// Relays stopper state and sends a message when stopper state changes.
FUNCTION_BLOCK FB_StopperWatcher
VAR_INPUT
END_VAR
VAR_OUTPUT
END_VAR
VAR_IN_OUT
	stCurrentBP : ST_BeamParams;
END_VAR
VAR
    i_StopperOutLS AT %I* : BOOL;
    i_StopperInLS AT %I* : BOOL;

    q_StopperOUT_Relay AT %Q* : BOOL;
    q_StopperIN_Relay AT %Q* : BOOL;

    Stopper : UINT;
    StopperName : STRING;
	{attribute 'instance-path'}
    {attribute 'noinit'}
    sPath    :    T_MaxString;

    // Logging
    fbLogMsg : FB_LogMessage := (
        eSubSystem := E_Subsystem.MPS);

    rtIn : R_TRIG;
    rtOut : R_TRIG;

	bInit: BOOL := TRUE;
END_VAR

IF bInit THEN
	fbLogMsg.sJson := F_PMPS_JSON(StopperName, sPath, 1000);
	bInit := FALSE;
END_IF


rtIn(CLK := i_StopperInLS);
rtOut(CLK := i_StopperOutLS);

IF rtIn.Q THEN
    fbLogMsg.sMsg := CONCAT(StopperName, ' moved IN');
    fbLogMsg();
ELSIF rtOut.Q THEN
    fbLogMsg.sMsg := CONCAT(StopperName, ' moved OUT');
    fbLogMsg();
END_IF

q_StopperOUT_Relay := i_StopperOutLS;
q_StopperIN_Relay := i_StopperInLS;

// Update current beam parameters
stCurrentBP.aVetoDevices[Stopper] := i_StopperInLS;

END_FUNCTION_BLOCK

// MajorComponents/Stoppers/FB_KVetoDevice
FUNCTION_BLOCK FB_KVetoDevice EXTENDS FB_VetoDevice
VAR_INPUT
END_VAR
VAR_OUTPUT
END_VAR
VAR
END_VAR

SUPER^(stCurrentBP:=SUPER^.stCurrentBP);

METHOD FB_init : BOOL
VAR_INPUT
	bInitRetains : BOOL; // if TRUE, the retain variables are initialized (warm start / cold start)
	bInCopyCode : BOOL;  // if TRUE, the instance afterwards gets moved into the copy code (online change)
    eVetoDeviceIN : K_Stopper := K_Stopper.DEFAULT;
    eVetoDeviceOUT : K_Stopper := K_Stopper.DEFAULT;
    sVetoDeviceName : STRING;
END_VAR
VetoDevice_IN := eVetoDeviceIN;
VetoDevice_OUT := eVetoDeviceOUT;
VetoDeviceName := sVetoDeviceName;
END_METHOD

END_FUNCTION_BLOCK

// MajorComponents/Stoppers/FB_VetoDevice
// Relays veto device state, updates current BP and sends a message when veto state changes.
FUNCTION_BLOCK FB_VetoDevice
VAR_INPUT
	i_bIn : BOOL;
	i_bOut : BOOL;
END_VAR
VAR_OUTPUT
    q_bIn : BOOL;
    q_bOut : BOOL;
END_VAR
VAR_IN_OUT
	stCurrentBP : ST_BeamParams;
END_VAR
VAR

    VetoDevice_IN : UINT := PMPS_GVL.MAX_VETO_DEVICES; // Veto device state array index
	VetoDevice_OUT : UINT := PMPS_GVL.MAX_VETO_DEVICES; // Veto device state array index
    
    VetoDeviceName : STRING;
	{attribute 'instance-path'}
    {attribute 'noinit'}
    sPath    :    T_MaxString;

    // Logging
        fbLogMsg : FB_LogMessage := (
            eSubSystem := E_Subsystem.MPS);
    
        rtIn : R_TRIG;
        rtOut : R_TRIG;
    ////////////////////////////////
    
	bInit: BOOL := TRUE;
END_VAR

IF bInit THEN
	fbLogMsg.sJson := F_PMPS_JSON(VetoDeviceName, sPath, 1000);
	bInit := FALSE;
END_IF

// Log
/////////////////////////////
    rtIn(CLK := i_bIn);
    rtOut(CLK := i_bOut);
    
    IF rtIn.Q THEN
        fbLogMsg.sMsg := CONCAT(VetoDeviceName, ' moved IN');
        fbLogMsg();
    ELSIF rtOut.Q THEN
        fbLogMsg.sMsg := CONCAT(VetoDeviceName, ' moved OUT');
        fbLogMsg();
    END_IF

// Relay
///////////////////////
    q_bIn := i_bIn;
    q_bOut := i_bOut;

// Update current beam parameters
/////////////////////////////////////
    stCurrentBP.aVetoDevices[VetoDevice_IN] := i_bIn;
    stCurrentBP.aVetoDevices[VetoDevice_OUT] := i_bOut;

END_FUNCTION_BLOCK

// MajorComponents/Stoppers/FB_LStopper
FUNCTION_BLOCK FB_LStopper EXTENDS FB_StopperWatcher
VAR_INPUT
END_VAR
VAR_OUTPUT
END_VAR
VAR_IN_OUT
END_VAR
VAR
END_VAR

SUPER^(stCurrentBP:=SUPER^.stCurrentBP);

METHOD FB_init : BOOL
VAR_INPUT
    bInitRetains : BOOL; // if TRUE, the retain variables are initialized (warm start / cold start)
    bInCopyCode : BOOL;  // if TRUE, the instance afterwards gets moved into the copy code (online change)
    eStopper : L_Stopper;
    sStopperName : STRING;
END_VAR
Stopper := eStopper;
StopperName := sStopperName;
END_METHOD

END_FUNCTION_BLOCK

// MajorComponents/FB_BPControlDevice
(*
Used to request a beam parameter set from EPICS.

Technically just one of these is needed in the entire
PMPS for a line.

*)
FUNCTION_BLOCK FB_BPControlDevice
VAR_INPUT
        (*  Requested pre-optic attenuation %  *)
        {attribute 'pytmc' := 'pv: ReqBP:Transmission
            io: o
			field: HOPR 1;
			field: LOPR 0;
			field: PREC 2;
        '}
        nTran : REAL := PMPS_GVL.TRANS_SCALING_FACTOR;
        (* Pulse-rate *)
        {attribute 'pytmc' := 'pv: ReqBP:Rate
            io: o
            field: EGU Hz
        '}
        nRate : UDINT := 10;
        (* Photon energy ranges *)
        {attribute 'pytmc' := 'pv: ReqBP:PhotonEnergyRanges
            io: o
            field: EGU eV'}
        {attribute 'displaymode' := 'binary'}
        neVRange : DWORD := 4294967295;
END_VAR
VAR_OUTPUT
END_VAR
VAR_IN_OUT
    Arbiter : FB_Arbiter;
END_VAR
VAR
    EpicsReqBP : ST_BeamParams;
    {attribute 'pytmc' := '
        pv: ReqBP:Apply
        io: o
    '}
    bApply : BOOL;

    nControlDeviceID : DWORD;
	sControlDeviceName: STRING:= 'BP Cntrl Dev';
    rtApply : R_TRIG;

END_VAR


EpicsReqBP.nTran := nTran;
EpicsReqBP.neVRange := neVRange;
EpicsReqBP.nRate := nRate;

rtApply(CLK:=bApply);
IF rtApply.Q THEN
    Arbiter.RemoveRequest(nControlDeviceID);
    Arbiter.AddRequest(nControlDeviceID, EpicsReqBP, sControlDeviceName);
    bApply := FALSE;
END_IF

METHOD FB_init : BOOL
VAR_INPUT
    bInitRetains : BOOL; // if TRUE, the retain variables are initialized (warm start / cold start)
    bInCopyCode : BOOL;  // if TRUE, the instance afterwards gets moved into the copy code (online change)
    nID : DWORD := PMPS_GVL.EXCLUDED_ASSERTION_ID;
END_VAR
nControlDeviceID:= nID;
END_METHOD

END_FUNCTION_BLOCK

// MajorComponents/FB_BPRequestor
(* BP Requestor
Elevates the BP request from an arbiter to PMPS_GVL.stRequestedBP
*)
FUNCTION_BLOCK FB_BPRequestor IMPLEMENTS I_HigherAuthority
VAR_INPUT
END_VAR
VAR_OUTPUT
    q_ReqBP : ST_BeamParams; // Arbitrated BP
END_VAR
VAR_IN_OUT
    Arbiter : FB_Arbiter;
    //FFO : FB_HardwareFFOutput;
END_VAR
VAR
    ReqBP : ST_BeamParams;
    nCohort : ULINT; // Current cohort, inc. 1 cycle after IO is updated
    nRequestCohort : ULINT; // Cohort number recorded at the time of the request.
END_VAR

Arbiter.ElevateRequest(THIS^); // Executes arbitration and retrieves ReqBP

IF nRequestCohort >= nCohort THEN
    // Update requested BP set
    q_ReqBP := ReqBP;
    // Note: we may do more here someday... perhaps all of the output control
    // will reside in here, and be solely controlled by this block. For now
    // I am going to adopt a flat management structure.
    // Start a new cohort
    nCohort := nCohort + 1;
END_IF

// Returns true when outputs to MPS are updated
METHOD CheckRequest : BOOL
VAR_INPUT
	nReqID	: DWORD;
END_VAR
VAR_INST
    xFirstTime : BOOL;
    nId : DWORD;
END_VAR
(* nRequestCohort will be < nCohort after output control
function blocks have been updated to reflect the new request
*)
CheckRequest := nRequestCohort < nCohort;
END_METHOD

METHOD RemoveRequest : BOOL
VAR_INPUT
	nReqID    :    DWORD; //StateID to remove
END_VAR
END_METHOD

METHOD RequestBP : BOOL
VAR_INPUT
	(*StateID of state requesting beam parameter set*)
	nReqID	: DWORD;
	(*Requested beam params*)
	stReqBP	: ST_BeamParams;
END_VAR
VAR_INST
    ReqID : DWORD;
    Registered : BOOL := FALSE;
END_VAR

// Check the request is coming from the same source we're used to
IF NOT Registered THEN
    ReqID := nReqID;
    Registered := TRUE;
END_IF
// log a complaint if false
RequestBP := ReqId = nReqId;

// Update internal BP request struct
ReqBP := stReqBP;

// Record current cohort

    nRequestCohort := nCohort;
END_METHOD

END_FUNCTION_BLOCK

// MajorComponents/FB_LinearGovernor

(* The governor is meant to check your work and keep you from making mistakes.

Checks:
Does your state match the device position and visa versa?
Are the beam parameters safe for the device state?
Did you properly assert the transition and final beam parameters?

*)
FUNCTION_BLOCK FB_LinearGovernor
VAR_INPUT
    i_stCurrentBeamParams    :    ST_BeamParams; //Link to global beam params
    i_xMPSOverride            :    BOOL; //True releases MPS limits after a delay
    i_xTransitionRequested    :    BOOL; //Set true to request a transition
    i_xResetMPSFault    :    BOOL; //Set true to clear MPS fault 
END_VAR
VAR_OUTPUT
     //True when governor has released restrictions
    q_xTransitionPermitted    :    BOOL;
    //Set if MC_Power has an error, or override mode is requested
    q_xFault    :    BOOL; 
    // Indicates override mode is active
    q_xMPSLimitsOverridden: BOOL;
END_VAR
VAR_IN_OUT
    stDevice    :    ST_Device; //The governed
    Arbiter    :    FB_Arbiter;
    FastFaultOutput    :    FB_HardwareFFOutput;
END_VAR
VAR
    mcPower    :    MC_Power;
    
    xActuatorPositiveEnable: BOOL;
    xActuatorNegativeEnable: BOOL;
    
    xMPSPositiveEnable    :    BOOL;
    xMPSNegativeEnable    :    BOOL;
    lrPosition: LREAL;
    
    lrLatchedTargetPosition    :    LREAL;
    lrLatchedTargetTolerance    :    LREAL;
    stLatchedTargetState    :    ST_DeviceStateExt;
    
    lrMPSUpperLimit: LREAL;
    lrMPSLowerLimit: LREAL;
    rtNewState: R_TRIG;
    xTransitionOK: BOOL;
    
    tonMPSOverrideMode    :    TON := (
        PT := T#5S
    );
    
    srMPSFault    :    SR;
    // Actuator out of bounds fault
    xActuatorOOB: BOOL;
    //Beam parameters out of spec
    xBeamParamsOOS: BOOL;
    //Beam parameters of currently latched state
    
    stLatchedBeamParams: ST_BeamParams;
    stTargetState: ST_DeviceStateExt;
    
    rtLatchNewState    :    R_TRIG;
    xInit: BOOL := TRUE;
    
    stInitDeviceState: ST_DeviceStateExt;
    // Indicates an error with initialization
    xInitFault: BOOL;
    // Indicates the state could not be found in the state table. There may be something wrong in the device state machine implementation or state table instantiation.
    xStateLookupError: BOOL;
    // A transition needs to be requested at least once before we start latching any state.
    xTransitionHasBeenRequested: BOOL := FALSE;
    ffBeamParamsOK : FB_FastFault;
    ffActuatorBoundsOK    :    FB_FastFault;
END_VAR


lrPosition := stDevice.stAxis.NcToPlc.ActPos; //Actuator position

stDevice.stAxis.ReadStatus();
//Init
(* The init strategy is:
If the device is restored and it's residing at the safe position,
no PMPS faults. *)
////////////////////////////////
    IF xInit THEN
        xInit := FALSE;
        //Use nSafeSate for initialization. 
        stDevice.StateTable.A_Lookup(key := stDevice.nSafeState);
        IF stDevice.StateTable.bOk THEN
            stInitDeviceState := F_DeviceState_To_DeviceStateExt(stDevice.StateTable.getValue, TRUE);
            xInitFault := FALSE;
        ELSE
            xInitFault := TRUE;
            stInitDeviceState.xValid := FALSE;
        END_IF
        lrLatchedTargetPosition := stInitDeviceState.rPosition;
        lrLatchedTargetTolerance := stInitDeviceState.rTolerance;
        stLatchedBeamParams := stInitDeviceState.stReqBeamParam;
    END_IF

// The governor will permit transitions once it verifies the transition assertion is active
// Note the governor does not verify the target state beam params are asserted, perhaps it should <TODO>
////////////////////////////////
    IF i_xTransitionRequested THEN
        xTransitionHasBeenRequested    := TRUE;
        
        xTransitionOK := Arbiter.CheckRequest( stDevice.stTransitionState.nStateRef) AND F_SafeBPCompare(i_stCurrentBeamParams, stDevice.stTransitionState.stReqBeamParam);
        
        //Set the target state for evaluation in further logic
        stdevice.StateTable.A_Lookup(key := stDevice.nTargetState);
        IF stDevice.StateTable.bOk THEN
            stTargetState := F_DeviceState_To_DeviceStateExt(stDevice.StateTable.getValue, TRUE);
            xStateLookupError := FALSE;
        ELSE
            xStateLookupError := TRUE;
            stTargetState.xValid := FALSE;
        END_IF
    ELSE
        xTransitionOK := FALSE;
    END_IF

(* Note about TransitionRequested

If TransitionRequested goes false during a transition, an MPS fault may be induced. This occurs
because the Actuator Out of Bounds fault will go back to using the original state limits, which
the axis may have already moved beyond.

To avoid this transient fault, make sure your device state machine is implemented such that the 
transition request to the governor block remains high until the target position is reached.
*)

//Determine if a transition is complete and latch the new state
(* A transition is complete when:

Axis at standstill.
Axis within tolerance.
No transition req.

Once these conditions are met, the MPS limits shall re-engage to restrict the
axis motion to the tolerance around the state position and the MPS fault monitors
shall evaluate based on the newly latched target state.
*)

rtLatchNewState(CLK := stDevice.stAxis.Status.StandStill AND
    lrPosition <= stTargetState.rPosition + stTargetState.rTolerance AND
    lrPosition >= stTargetState.rPosition - stTargetState.rTolerance AND
    NOT i_xTransitionRequested AND xTransitionHasBeenRequested);
    
IF rtLatchNewState.Q THEN
    lrLatchedTargetPosition := stTargetState.rPosition;
    lrLatchedTargetTolerance := stTargetState.rTolerance;
    stLatchedBeamParams := stTargetState.stReqBeamParam;
    stLatchedTargetState := stTargetState;
END_IF

//Let other blocks know the governor won't interfer with transitions
q_xTransitionPermitted := xTransitionOK;

//Adjust limit ranges based on active state and current target
IF xTransitionOK THEN
    //Extend range to include target state
    lrMPSUpperLimit := MAX(lrMPSUpperLimit, stTargetState.rPosition + stTargetState.rTolerance);
    lrMPSLowerLimit := MIN(lrMPSLowerLimit, stTargetState.rPosition - stTargetState.rTolerance);
ELSE
    //Calculate the limit positions for MPS based on current state
    lrMPSUpperLimit := lrLatchedTargetPosition + lrLatchedTargetTolerance;
    lrMPSLowerLimit := lrLatchedTargetPosition - lrLatchedTargetTolerance;
END_IF


//MPS override
(* In override mode, the device will be free to move anywhere within it's travel range *)
//Permit motion after a small delay
tonMPSOverrideMode(IN:=i_xMPSOverride OR stDevice.xOverrideMPSLimits, Q=>q_xMPSLimitsOverridden);

//Virtual limit switch evaluation
xActuatorPositiveEnable    := stDevice.i_xHiLim AND lrPosition <= stDevice.lrUpperPositionLimit;
xActuatorNegativeEnable    := stDevice.i_xLoLim AND lrPosition >= stDevice.lrLowerPositionLimit;

//Evaluate MPS limit states
xMPSPositiveEnable := lrPosition <= lrMPSUpperLimit;
xMPSNegativeEnable := lrPosition >= lrMPSLowerLimit;

//Final Limit switch evaluation
mcPower.Enable_Positive := xActuatorPositiveEnable AND (tonMPSOverrideMode.Q OR xMPSPositiveEnable);
mcPower.Enable_Negative := xActuatorNegativeEnable AND (tonMPSOverrideMode.Q OR xMPSNegativeEnable);

mcPower(
    Axis := stDevice.stAxis,
    Enable := stDevice.xEnable //link to device enable <TODO>
);



//MPS Faults
//Fault if the beam is unsafe for current state
ffBeamParamsOK(i_xOK:=F_SafeBPCompare(i_stCurrentBeamParams, stLatchedBeamParams), 
                i_xReset:=i_xResetMPSFault,
                io_fbFFHWO := FastFaultOutput);

//Fault if the position is outside of the permitted range
ffActuatorBoundsOK(i_xOK := (lrPosition <= lrMPSUpperLimit AND lrPosition >= lrMPSLowerLimit), 
                    i_xReset:=i_xResetMPSFault,
                io_fbFFHWO := FastFaultOutput);


    
//Collect all other faults
q_xFault := NOT ffBeamParamsOK.o_xFFLine OR
    NOT ffActuatorBoundsOK.o_xFFLine OR
    mcPower.Error    OR
    i_xMPSOverride    OR
    xInitFault;

//Any faults trip the fast fault line for this FB    
//FastFaultOutput.CheckIn(NOT q_xFault);

END_FUNCTION_BLOCK

// MajorComponents/FB_RateFromEPICS
FUNCTION_BLOCK FB_RateFromEPICS

(*
enum MPSBeamRates {
    MPSRateInvalid            =  0,
    MPSRate0Hz                =  1,
    /* Previously used 2 and 3 for single shot and burst */
    MPSRate1Hz                =  4,
    MPSRate10Hz               =  5,
    MPSRate30Hz               =  6,
    MPSRate60Hz               =  7,
    MPSRate120Hz              =  8,
    MPSRateUnknown            =  9,
    MPSRateSingleShot         = 10,
    MPSRateBurstMode          = 11,
    MPSRateBurstModeNotActive = 12,
    MPSNumberOfBeamRates      = 13,
    MPSRateBurstInvalid       = 14
}
*)

VAR_IN_OUT
	BP : ST_BeamParams;
    fbBYKIK_Rate : FB_LREALFromEPICS;
	FFO : FB_HardwareFFOutput;
END_VAR
VAR_OUTPUT
	xError : BOOL;
END_VAR
VAR

	
	eMPSRate : E_MPSBeamRates;
	
	ffRateReadBack : FB_FastFault := (
		i_DevName := 'Arbiter',
		i_Desc := 'Issue with rate readback from Accelerator. Gateway or EPICS connection. Must be fixed.',
		i_TypeCode := 16#203,
		i_xAutoReset:=True);
END_VAR
VAR CONSTANT
	cFailSafeRate : UDINT := 1000001;
END_VAR

fbBYKIK_Rate();

IF fbBYKIK_Rate.bValid THEN
	eMPSRate := LREAL_TO_UINT(fbBYKIK_Rate.fValue);
ELSE
	eMPSRate := E_MPSBeamRates.MPSRateInvalid;
END_IF

CASE eMPSRate OF
	MPSRateInvalid:
		BP.nRate := cFailSafeRate;
	MPSRate0Hz:
		BP.nRate := 0;
	MPSRate1Hz:
		BP.nRate := 1;
	MPSRate10Hz:
		BP.nRate := 10;
	MPSRate30Hz:
		BP.nRate := 30;
	MPSRate60Hz:
		BP.nRate := 60;
	MPSRate120Hz:
		BP.nRate := 120;
	MPSRateUnknown:
		BP.nRate := cFailSafeRate;
	
ELSE
	BP.nRate := cFailSafeRate;
END_CASE

ffRateReadback(i_xOK:=fbBYKIK_Rate.bValid, io_fbFFHWO:=FFO);

BP.xValid R= NOT fbBYKIK_Rate.bValid OR
			eMPSRate = MPSRateUnknown OR
			eMPSRate = MPSRateInvalid;

END_FUNCTION_BLOCK

// TestComponents/FB_Arbiter_Test
{attribute 'call_after_init'}
FUNCTION_BLOCK FB_Arbiter_Test EXTENDS TcUnit.FB_TestSuite
VAR_INPUT
END_VAR
VAR_OUTPUT
END_VAR
VAR
END_VAR

Arbitration();
RequestCheckRemoveBP();
FullArbitrationStack();
StackArbiters();
RemoveReq();
DoS();

METHOD ArbiterCapacity
VAR_INPUT
END_VAR
VAR   
    nId    :    DWORD := 1;
    stReq    :    ST_BeamParams := (nTran:=12);
    
    nRandID : DWORD;
    testReq : ST_BeamParams := (neVRange := 16#FFEE, nRate:=33);
    
    idx : DWORD;

END_VAR
VAR_INST
    fbArbCapacityTest    :    FB_Arbiter(1);

    Cycle : INT := 0;
    
    CycleLimit : INT := 20;
    
END_VAR
VAR CONSTANT
    SysID : DWORD := 42;
END_VAR

TEST('Arbiter Capcity');
    // Fill the arbiter
    FOR idx := 1 TO PMPS_PARAM.MAX_ASSERTIONS DO
        fbArbCapacityTest.AddRequest(nReqID := idx, stReqBP := testReq, sDevName:= CONCAT('Device #', TO_STRING(idx)));
    END_FOR

TEST_FINISHED();
END_METHOD

METHOD Arbitration
VAR_INPUT
END_VAR
VAR
    
     nTranReqID    :    UDINT    := 1;
    stAttReqBP    :    ST_BeamParams := PMPS_GVL.cstFullBeam;
    
    nPPEReqID    :    UDINT    := 2;
    stPPEReqBP    :    ST_BeamParams := PMPS_GVL.cstFullBeam;
    
    nEVReqID    :    UDINT    := 3;
    stEVReqBP    :    ST_BeamParams := PMPS_GVL.cstFullBeam;
    
    nRateReqID    :    UDINT    := 4;
    stRateReqBP    :    ST_BeamParams := PMPS_GVL.cstFullBeam;
    
    stArbitratedBP    :    ST_BeamParams;
    stExpectedBP    :    ST_BeamParams := PMPS_GVL.cstFullBeam;;
END_VAR
VAR_INST
    fbArbiter    :    FB_Arbiter(1);
END_VAR
TEST('Arbitration');

stAttReqBP.nTran := 0.50;
stEVReqBP.neVRange := 2#1111_1111_1111_1111_1111_1100_1111_1111;
stRateReqBP.nRate := 10;

stExpectedBP.nTran     :=     stAttReqBP.nTran;
stExpectedBP.neVRange := stEVReqBP.neVRange;
stExpectedBP.nRate := stRateReqBP.nRate;

//Load arbiter with beam parameter sets
AssertTrue(fbArbiter.AddRequest(nTranReqID, stAttReqBP, sDevName:= 'Device' ),
                    'Safest attenuation request failed to load');
                    
//Load arbiter with beam parameter sets
AssertTrue(fbArbiter.AddRequest(nPPEReqID, stPPEReqBP, sDevName:= 'Device'),
                    'Safest PPE request failed to load');
                    
//Load arbiter with beam parameter sets
AssertTrue(fbArbiter.AddRequest(nEVReqID, stEVReqBP, sDevName:= 'Device'),
                    'Safest stEVReqBP request failed to load');
                    
//Load arbiter with beam parameter sets
AssertTrue(fbArbiter.AddRequest(nRateReqID, stRateReqBP, sDevName:= 'Device'),
                    'Safest stRateReqBP request failed to load');

stArbitratedBP := fbArbiter.GetArbitratedBP();

AssertFalse(F_DifferentBeamParams(stExpectedBP, stArbitratedBP),
                'Arbitrated BP does not match expected.');

TEST_FINISHED();
END_METHOD

METHOD DoS
VAR
    

    
    nOrigReqID : UDINT := 30;
    nSecondReqID : UDINT := 35;
    
    nPeskyReqID : UDINT := 40;
    
    
END_VAR
VAR_INST
    DosArb : FB_Arbiter(20);
    
    DummyHA : FB_DummyHA := (ReqAcknowledged:=FALSE); // Set req ack false to start so we can control when it is verified
    nTimeoutCounter : UINT;
    bInit : BOOL;
    bSecond : BOOL;
    eDosTestCases : E_ArbDosTestStates;
END_VAR
VAR CONSTANT
        nTimeoutCounterMAX : UINT := 50;
        nWaitCount : UINT := 10;
        nWait2ndCount : UINT := nWaitCount + 5;
END_VAR
TEST('DoS');

CASE eDosTestCases OF
    E_ArbDosTestStates.Init: // Init, first request
        DosArb.AddRequest(nOrigReqID, PMPS_GVL.cst0RateBeam, sDevName:= 'Device');
        eDosTestCases := E_ArbDosTestStates.SecondReq;
        
    E_ArbDosTestStates.SecondReq: // Add second request
        DosArb.AddRequest(nSecondReqID, PMPS_GVL.cst0RateBeam, sDevName:= 'Device');
        eDosTestCases := E_ArbDosTestStates.WaitForAck;
        
    E_ArbDosTestStates.WaitForAck:
        IF nTimeoutCounter > nWaitCount THEN
            DummyHA.ReqAcknowledged := TRUE;
            eDosTestCases := E_ArbDosTestStates.WaitFor2ndAck;
		END_IF
    
    E_ArbDosTestStates.WaitFor2ndAck:
        DummyHA.ReqAcknowledged := False;
        IF nTimeoutCounter > nWait2ndCount THEN
            DummyHA.ReqAcknowledged := TRUE;
            eDosTestCases := E_ArbDosTestStates.RunAsserts;
		END_IF
    
END_CASE

DosArb.ElevateRequest(DummyHA);

// Pesky request always adding and removing
DosArb.RemoveRequest(nPeskyReqID);
DosArb.AddRequest(nPeskyReqID, PMPS_GVL.cst0RateBeam, sDevName:= 'Device');


nTimeoutCounter := nTimeoutCounter + 1;

IF nTimeoutCounter > nTimeoutCounterMAX or eDosTestCases = E_ArbDosTestStates.RunAsserts THEN 
    AssertTrue(DosArb.CheckRequest(nOrigReqID), 'Original request still not accepted');
    AssertTrue(DosArb.CheckRequest(nSecondReqID), 'Second request still not accepted'); 
   
    TEST_FINISHED_NAMED('DoS');
END_IF
END_METHOD

METHOD FullArbitrationStack
VAR_INPUT
END_VAR
VAR   
    nId    :    DWORD := 1;
    stReq    :    ST_BeamParams := (nTran:=12);
	
	nIdDoS : DWORD := 13;
	stDoSReq : ST_BeamParams := PMPS_GVL.cstFullBeam;
END_VAR
VAR_INST
    fbArbiter    :    FB_Arbiter(1);
    
    fbHigherArb : FB_Arbiter(2);
    
    fbSubSysToArb : FB_SubSysToArbiter_IO; // Subsystem interface with beamline arbiter PLC
    pBPR : POINTER TO ST_BeamParams_IO;
    
    fbArbToSubSys : FB_ArbiterToSubSys_IO := (RequestingSystemID:=42); // Beamline arbiter PLC interface with subsystems
    pBPC : POINTER TO ST_BeamParams_IO;
    
    fbBPR : FB_BPRequestor; // Use in the arbiter PLC to apply an arbitrated beam parameter set to the accelerator interface
    
    FFO : FB_HardwareFFOutput; // Dummy FFO not important for these tests

    Cycle : INT := 0;
    
    CycleLimit : INT := 20;
    
END_VAR
VAR CONSTANT
    SysID : DWORD := 42;
END_VAR
// This simulates a synchronous cycle between the subsystem and arbiter PLC cycles. Ie. phase is locked, and cycle time is the same. This is not always the case, so these tests should be 
// trusted with a grain of salt.

TEST('FullStack');



CASE Cycle OF

0: 
    IF NOT fbArbiter.CheckRequestInPool(nID) THEN
        AssertTrue(fbArbiter.AddRequest(nId, stReq,'Device'), 'Arbiter returned false from AddRequest'); // some device asking its local arbiter for some beam parameters
    END_IF  
    
    TEST('JustEnteredRequest');
    AssertFalse(fbArbiter.CheckRequest(nId),
        'Check should fail. Request not arbitrated yet.');
    TEST_FINISHED();
   
8000:
    TEST_FINISHED_NAMED('FullStack');   
    
END_CASE 


TEST('VerifyBPRHasBP');
IF fbHigherArb.CheckRequest(SysID) THEN
    AssertFalse(F_DifferentBeamParams(stReq, fbBPR.q_ReqBP),
        'Beam parameters not fully propagated to BPR at highest level');
        TEST_FINISHED_NAMED('VerifyBPRHasBP');
END_IF

TEST('ArbToSubsysPropagation');
IF fbArbToSubSys.nActiveCohort = fbArbToSubSys.nRequestedCohort 
    AND fbArbToSubSys.nActiveCohort <> 0 THEN
    AssertTrue(fbHigherArb.CheckRequest(SysID),
        'Active cohort = Requested cohort before higher arbiter confirmed request was active');
    TEST_FINISHED_NAMED('ArbToSubsysPropagation');
END_IF

TEST('SubsysToArbPropagation');
IF fbArbiter.CheckRequest(nId) THEN
    AssertTrue(fbSubSysToArb.nActiveCohort >= fbSubSysToArb.nRequestCohort,
        'Request validated before higher level confirmation');
    TEST_FINISHED_NAMED('SubsysToArbPropagation');
END_IF


TEST('VerifyIncludedAtAllLevels');
IF fbArbiter.CheckRequest(nId) THEN
    AssertTrue(fbHigherArb.CheckRequest(fbArbToSubSys.RequestingSystemID), 'HigherArb is not yet included in arbitration');
    AssertTrue(fbSubSysToArb.CheckRequest(fbArbiter.nLowerAuthorityID), 'Local Arb is not yet included in arbitration');
    TEST_FINISHED_NAMED('VerifyIncludedAtAllLevels');
END_IF
      
    
///////////////////////////////////////
//Sub system cycle
fbSubSysToArb(Arbiter := fbArbiter, fbFFHWO := FFO);
//END of sub system cycle
///////////////////////////////////////

//Ethercat transfer simulation
// Transfer of requested BP to arbiter PLC
pBPR := ADR(fbArbToSubSys.i_RequestedBP);
pBPR^ := fbSubSysToArb.q_stRequestedBP;

// Transfer of current BP to sub system PLC
pBPC := ADR(fbSubSysToArb.i_stCurrentBP);
pBPC^ := fbArbToSubSys.o_CurrentBP;

//////////////////////////////////////
//Start of arbiter plc cycle
//Arb io collects sub system status
fbArbToSubSys(Arbiter := fbHigherArb, fbFFHWO := FFO); // This is making a request in the higher arb
//BPR collects arbiter summation
fbBPR(Arbiter := fbHigherArb); // This is getting the arbitrated BP




IF CycleLimit > Cycle THEN
    Cycle := Cycle + 1;
ELSE 
    Cycle := 8000;
END_IF
END_METHOD

METHOD RemoveReq
VAR
    
    Arb : FB_Arbiter(20);
    
    DummyHA : FB_DummyHA;
    
    Result : BOOL;
    
END_VAR

Arb.AddRequest(30, PMPS_GVL.cst0RateBeam, 'Device');

Arb.ElevateRequest(DummyHA);

TEST('Remove Req');
    Result := Arb.RemoveRequest(77);
    
    AssertFalse( Result, 'RemoveReq returned true, with nothing to remove');
    AssertFalse( Arb.bStartNewAckRequest , 'StartNewAckRequest is set. Something is wrong');
    
TEST_FINISHED();
END_METHOD

METHOD RequestCheckRemoveBP
VAR_INPUT
END_VAR
VAR
    
    nId    :    DWORD := 1;
    stReq    :    ST_BeamParams;
END_VAR
VAR_INST
    fbArbiter    :    FB_Arbiter(1);
END_VAR
TEST('RequestBP');
AssertTrue(fbArbiter.AddRequest(nId, stReq, 'Device'),
    'Request failed');

TEST_FINISHED();
    
TEST('DuplicateID');
AssertFalse(fbArbiter.AddRequest(nId, stReq, 'Device'),
    'Duplicate request accepted, not good.');

TEST_FINISHED();
    
TEST('CheckBP');
AssertFalse(fbArbiter.CheckRequest(nId),
    'Check should fail. Request not arbitrated yet.');
TEST_FINISHED();

TEST('CheckBPArbitrated');
WRITE_PROTECTED_ULINT(ADR(fbArbiter.nActiveCohort), fbArbiter.nNextCohort);
AssertTrue(fbArbiter.CheckRequest(nId),
    'Check should pass.');

TEST_FINISHED();      
    
TEST('IDDoesNotExist');
 
AssertFalse(fbArbiter.CheckRequest(nId+1),
    'Check returned true when ID does not exist');

TEST_FINISHED();
    
TEST('RemoveBP');
AssertTrue(fbArbiter.RemoveRequest(nId),
    'Remove failed');
AssertFalse(fbArbiter.CheckRequest(nId),
    'Remove did not remove request');
    
TEST_FINISHED();

TEST('NoRequestsFullBeam');

AssertFalse(F_DifferentBeamParams(fbArbiter.GetArbitratedBP(), PMPS_GVL.cstFullBeam), 'Arbitrated beam should be full with all requests removed');

TEST_FINISHED();
END_METHOD

METHOD StackArbiters
VAR_INPUT
END_VAR
VAR   
    nId    :    DWORD := 1;
    stReq    :    ST_BeamParams := (nTran:=12);
END_VAR
VAR_INST
    fbArbiter    :    FB_Arbiter(1);
    
    fbHigherArb : FB_Arbiter(2);
	
	ArbBP : ST_BeamParams;

    Cycle : INT := 0;
    
    CycleLimit : INT := 20;
    
END_VAR
VAR CONSTANT
    SysID : DWORD := 42;
END_VAR

TEST('StackingArbiters');
fbArbiter.AddRequest(nReqID:=nId, stReqBP:=stReq, sDevName :='Device');

fbArbiter.ElevateRequest(fbHigherArb);

ArbBP := fbHigherArb.GetArbitratedBP();

AssertTrue(ArbBP.nTran = 12, 'We should see the transmission number here');

TEST_FINISHED();
END_METHOD

END_FUNCTION_BLOCK

// TestComponents/FB_ArbToSubsys_Test
{attribute 'call_after_init'}
FUNCTION_BLOCK FB_ArbToSubsys_Test EXTENDS TcUnit.FB_TestSuite
VAR_INPUT
END_VAR
VAR_OUTPUT
END_VAR
VAR
END_VAR

BasicFunction();

METHOD BasicFunction
VAR_INPUT
END_VAR
VAR CONSTANT
    SysID : DWORD := 42;
END_VAR
VAR   
    nId    :    DWORD := 1;
    stReq    :    ST_BeamParams := (nTran:=12);
END_VAR
VAR_INST
    fbArbiter    :    FB_Arbiter(1);
    
    pBPR : POINTER TO ST_BeamParams_IO;
    
    stBPRIO : ST_BeamParams_IO := (
        nCohortInt := 1,
        nTran := 35); // Simulates subsystem BP request
    
    fbArbToSubSys : FB_ArbiterToSubSys_IO := (RequestingSystemID:=42); // Beamline arbiter PLC interface with subsystems
    pBPC : POINTER TO ST_BeamParams_IO;
    
    fbBPR : FB_BPRequestor; // Use in the arbiter PLC to apply an arbitrated beam parameter set to the accelerator interface
    
    FFO : FB_HardwareFFOutput; // Dummy FFO not important for these tests

    Cycle : INT := 0;
    
    CycleLimit : INT := 20;
    
END_VAR

// Simulate an initial cycle with no new requests coming in
fbBPR(Arbiter:=fbArbiter);
fbArbToSubSys(Arbiter:=fbArbiter, fbFFHWO:=FFO);

TEST('Init');
TEST_FINISHED();

//Ethercat transfer simulation
// Transfer of requested BP to arbiter PLC
pBPR := ADR(fbArbToSubSys.i_RequestedBP);
pBPR^ := stBPRIO;

///////////////////////////////////////
//Sub system cycle
fbBPR(Arbiter:=fbArbiter);
fbArbToSubSys(Arbiter:=fbArbiter, fbFFHWO:=FFO);
//END of sub system cycle
///////////////////////////////////////


TEST('New request');
    AssertTrue(fbArbToSubSys.nRequestedCohort = fbArbToSubSys.i_RequestedBP.nCohortInt, 'ReqCohort and qBP Cohort do not match, and they should');
    AssertTrue(fbArbiter.CheckRequestInPool(SysID), 'ArbToSubSys request should be in arbiter pool now');
    AssertTrue(fbArbToSubSys.nActiveCohort = 0, 'Active cohort should remain the initial value until the current request is active in higher arbitration');
    AssertTrue(fbArbToSubSys.o_CurrentBP.nCohortInt = fbArbToSubSys.nActiveCohort, 'Cohort being sent to sub system remains unincremented');
TEST_FINISHED_NAMED('New request');
    

///////////////////////////////////////
//Sub system cycle
fbBPR(Arbiter:=fbArbiter);
fbArbToSubSys(Arbiter:=fbArbiter, fbFFHWO:=FFO);
//END of sub system cycle
///////////////////////////////////////

///////////////////////////////////////
//Sub system cycle
fbBPR(Arbiter:=fbArbiter);
fbArbToSubSys(Arbiter:=fbArbiter, fbFFHWO:=FFO);
//END of sub system cycle
///////////////////////////////////////

///////////////////////////////////////
//Sub system cycle
fbBPR(Arbiter:=fbArbiter);
fbArbToSubSys(Arbiter:=fbArbiter, fbFFHWO:=FFO);
//END of sub system cycle
///////////////////////////////////////

TEST('Request has become active');
    AssertTrue(fbArbToSubSys.nRequestedCohort = fbArbToSubSys.nActiveCohort, 'ReqCohort and qBP Cohort do not match, and they should');
    AssertTrue(fbArbiter.CheckRequest(SysID), 'ArbToSubSys request should be in arbiter pool now');
    AssertTrue(fbArbToSubSys.nActiveCohort = stBPRIO.nCohortInt, 'Active cohort should remain the initial value until the current request is active in higher arbitration');
    AssertTrue(fbBPR.q_ReqBP.nTran = stBPRIO.nTran, 'BPR and requested BP should match');
TEST_FINISHED_NAMED('Request has become active');
END_METHOD

END_FUNCTION_BLOCK

// TestComponents/FB_AttenuatorSimulator
FUNCTION_BLOCK FB_AttenuatorSimulator
VAR_INPUT
    i_rRequestedAttenuation    :    REAL;
    i_stBPReadback    :    ST_BeamParams;
END_VAR
VAR_OUTPUT
    q_xFault    :    BOOL;
    q_rCurrentAttenuation    :    REAL;
END_VAR
VAR_IN_OUT
    Arbiter    :    FB_Arbiter; //Higher level arbiter from which upstream attenuation can be requested
END_VAR
VAR
    tonDelay    :    TON := (
        PT := T#3S
        );
END_VAR

// Really basic delay
tonDelay(IN := i_rRequestedAttenuation <> q_rCurrentAttenuation);

IF tonDelay.Q THEN
    q_rCurrentAttenuation := i_rRequestedAttenuation;
END_IF

END_FUNCTION_BLOCK

// TestComponents/FB_BPTM_Test
{attribute 'call_after_init'}
FUNCTION_BLOCK FB_BPTM_Test EXTENDS TcUnit.FB_TestSuite
VAR_INPUT
END_VAR
VAR_OUTPUT
END_VAR
VAR
END_VAR
VAR CONSTANT
    BPTM_ARR : UDINT := PMPS_PARAM.MAX_ASSERTIONS;
    cCycle : UINT := 20; // How many cycles does it take to complete a BPTM
END_VAR

BPTMBasicFunction();
InterruptAtAllSteps();
FullArbError();

METHOD BPTMBasicFunction
VAR_INPUT
END_VAR
VAR    
    //Final and transition assertions
    nTransitionID    :    UDINT := 1;
    stTransitionAssertion    :    ST_BeamParams := (nRate := 10);
    
    nReqID    :    UDINT    := 2;
    stReqAssertion    :    ST_BeamParams := (nTran := 0.2);
    
END_VAR
VAR_INST
    fbBPTM_TestBasicFunction    :    BeamParameterTransitionManager;
    fbArbiter    :    FB_Arbiter(1);
    ffo : FB_HardwareFFOutput;
    fbSubSysIO : FB_DummyArbIO;
    xFirstPass    :    BOOL := TRUE;
    eTestStep: E_BPTMTestStates := E_BPTMTestStates.Init;
END_VAR

// Completes arbiter request elevation process
// Necessary for CheckRequest to return true, ever
    fbBPTM_TestBasicFunction(
        fbArbiter := fbArbiter,
        );

fbSubSysIO(LA := fbArbiter, FFO := ffo);

// Note: this struct may also be (over)written to in the tests below, specifically rate.
fbBPTM_TestBasicFunction.stCurrentBeamParameters := fbSubSysIO.q_stSimulatedBPReadback;

CASE eTestStep OF

E_BPTMTestStates.Init:
    
    TEST('BPTMTest');
    eTestStep := E_BPTMTestStates.WaitingForBeam;

E_BPTMTestStates.WaitingForBeam:
    TEST('BPTM Waits for Beam');
    
    fbBPTM_TestBasicFunction.i_TransitionAssertionID := nTransitionID;
    fbBPTM_TestBasicFunction.i_stTransitionAssertion := stTransitionAssertion;
    
    fbBPTM_TestBasicFunction.i_nRequestedAssertionID := nReqID;
    fbBPTM_TestBasicFunction.i_stRequestedAssertion := stReqAssertion;
    
    IF fbBPTM_TestBasicFunction.eBPTMState = E_BPTMState.WaitForBP AND 
        NOT fbBPTM_TestBasicFunction.xEntry THEN
    
        AssertTrue(fbArbiter.CheckRequestInPool(nTransitionID), 'Arbiter did not accept BPTM transition assertion');
        
        AssertTrue(fbArbiter.CheckRequestInPool(nReqID), 'Arbiter did not accept BPTM transition assertion');
                
        AssertFalse(fbBPTM_TestBasicFunction.q_xTransitionAuthorized,
            'Transition should not be authorized until requests are in and beam is ready');
            
        AssertTrue(fbBPTM_TestBasicFunction.bBusy, 'Busy should be true here');
        AssertFalse(fbBPTM_TestBasicFunction.bDone, 'Done should be false');
        AssertFalse(fbBPTM_TestBasicFunction.bError, 'Error should be false here');
            
        TEST_FINISHED_NAMED('BPTM Waits for Beam');
        
        eTestStep := E_BPTMTestStates.Transitioning;
    END_IF    
    
    
E_BPTMTestStates.Transitioning:
    TEST('BPTM Authorizes Transition');

    fbBPTM_TestBasicFunction.stCurrentBeamParameters.nRate := 0; // satisfies the transition request   
    
    IF fbBPTM_TestBasicFunction.eBPTMState = E_BPTMState.Transitioning AND
        NOT fbBPTM_TestBasicFunction.xEntry THEN
    
        AssertTrue(fbArbiter.CheckRequest(nTransitionID),
            'Transition assertion should be in arbiter');
        
        AssertTrue(fbArbiter.CheckRequest(nReqID),
            'Final assertion should be in arbiter');
            
        AssertTrue(fbBPTM_TestBasicFunction.q_xTransitionAuthorized,
            'Transition should be authorized at this point.');
            
        AssertEquals(nReqID, fbBPTM_TestBasicFunction.nCurrentAssertionID,
            'nCurrentAssertionID not set.');
    
        TEST_FINISHED_NAMED('BPTM Authorizes Transition');
        
        eTestStep := E_BPTMTestStates.WaitingForFinalAssertion;
    END_IF

E_BPTMTestStates.WaitingForFinalAssertion:
    TEST('BPTM Waits for final BP');
    
    fbBPTM_TestBasicFunction.i_xDoneMoving := TRUE;
    
    IF fbBPTM_TestBasicFunction.eBPTMState = E_BPTMState.WaitForFinalBP THEN
        
        AssertTrue(fbArbiter.CheckRequest(nTransitionID),
        'Transition assertion should be in arbiter');  
        
        TEST_FINISHED_NAMED('BPTM Waits for final BP');
        
        eTestStep := E_BPTMTestStates.CleaningUp;
    END_IF    
    
E_BPTMTestStates.CleaningUp:

    fbSubSysIO.AutoUpdateBP := TRUE;

    TEST('Cleaning up');
    
    IF fbBPTM_TestBasicFunction.eBPTMState = E_BPTMState.Done THEN
        
        AssertFalse(fbArbiter.CheckRequestInPool(nTransitionID), 'Transition req should be removed from arb now');
        
        eTestStep := E_BPTMTestStates.Done; 
        
        TEST_FINISHED_NAMED('Cleaning up');
	END_IF

E_BPTMTestStates.Done:

    
    AssertTrue(fbBPTM_TestBasicFunction.bDone, 'Done should be set');
    AssertFalse(fbBPTM_TestBasicFunction.bError, 'Error should be cleared');
    AssertFalse(fbBPTM_TestBasicFunction.bBusy, 'Busy should be false');
    
    TEST_FINISHED_NAMED('BPTMTest');    
    
END_CASE
END_METHOD

// Simulate error due to full arbiter
METHOD FullArbError
VAR_INPUT
END_VAR
VAR    
    //Final and transition assertions
    nTransitionID    :    UDINT := 1000;
    stTransitionAssertion    :    ST_BeamParams :=  ( nTran := 0, neVRange := 0, nRate  := 0);//PMPS_GVL.cstSafeBeam;
    
    nReqID    :    UDINT    := 2000;
    stReqAssertion    :    ST_BeamParams := ( nTran := 0, neVRange := 0, nRate  := 0);//PMPS_GVL.cstSafeBeam;
    
    idx : UDINT;
    
    nRandID : DWORD;
    testReq : ST_BeamParams := (neVRange := 16#FFEE, nRate:=33);
    
END_VAR
VAR_INST
    fbBPTM_TestFullArb    :    BeamParameterTransitionManager;
    fbArbFullErr    :    FB_Arbiter(1);
    ffo : FB_HardwareFFOutput;
    fbSubSysIO : FB_DummyArbIO;
    fbBPR :  FB_BPRequestor;
    xFirstPass    :    BOOL := TRUE;
    eTestStep: E_BPTMTestStates := E_BPTMTestStates.Init;
    tonRetryTimeout : TON := (PT:=T#5s);
    entryToRetry : bool := true;
    fbRand : DRAND := (Seed :=1);
END_VAR
CASE eTestStep OF

E_BPTMTestStates.Init:
    
    TEST('BPTMErrorFullArb');
    
    // Fill the arbiter
    FOR idx := 1 TO PMPS_PARAM.MAX_ASSERTIONS // this fills the arbiter
                    - fbBPTM_TestFullArb.cReqArbCapacity + 1 DO // but test just one over the allowed amount
        fbArbFullErr.AddRequest(nReqID := idx, stReqBP := testReq, sDevName :='Device');
    END_FOR
    
    fbSubSysIO.AutoUpdateBP := TRUE;
    
    AssertTrue(PMPS_PARAM.MAX_ASSERTIONS - fbArbFullErr.nEntryCount < fbBPTM_TestFullArb.cReqArbCapacity,
        'Arbiter is not full enough, rest of tests will be invalid'); 
    
    eTestStep := E_BPTMTestStates.Error;

E_BPTMTestStates.Error:
    
    TEST('BPTM Full Error');

    IF fbBPTM_TestFullArb.bError THEN
        
        AssertTrue(fbBPTM_TestFullArb.bError AND fbBPTM_TestFullArb.nErrId = PMPS_CODES.NoRoomInArb,
            'Incorrect error response from full arbiter.');
            
        TEST_FINISHED_NAMED('BPTM Full Error');
        
        eTestStep := E_BPTMTestStates.Retry;
        
	END_IF
    
E_BPTMTestStates.Retry:
    
    TEST('Test Retry Post Failed Final');
    
    // Clear the arbiter
    if entryToRetry THEN
        FOR idx := 1 TO PMPS_PARAM.MAX_ASSERTIONS + 1 DO
            fbArbFullErr.RemoveRequest(idx);
        END_FOR
        entryToRetry := FALSE;
    END_IF
    
    // Push the retry button
    fbBPTM_TestFullArb.bRetry := TRUE;
    
    tonRetryTimeout(IN:=TRUE);
    
    IF tonRetryTimeout.Q OR fbBPTM_TestFullArb.q_xTransitionAuthorized THEN
        AssertTrue(fbBPTM_TestFullArb.q_xTransitionAuthorized, 'Transition should have been authorized by now');
        AssertTrue(fbArbFullErr.CheckRequest(nTransitionID), 'Transition ID is missing from arbiter while transition is authorized');
        AssertTrue(fbArbFullErr.CheckRequest(nReqID), 'Final ID is missing from arbiter while transition is authorized');
        
        TEST_FINISHED_NAMED('Test Retry Post Failed Final');
        
        eTestStep := E_BPTMTestStates.CleaningUp;
	END_IF

E_BPTMTestStates.CleaningUp:
    TEST_FINISHED_NAMED('BPTMErrorFullArb');    
    
END_CASE

fbBPTM_TestFullArb(
    fbArbiter := fbArbFullErr,
    i_TransitionAssertionID := nTransitionID,
    i_stTransitionAssertion := stTransitionAssertion,
    
    i_nRequestedAssertionID := nReqID,
    i_stRequestedAssertion := stReqAssertion,
    
    stCurrentBeamParameters := fbSubSysIO.q_stSimulatedBPReadback,
);

fbSubSysIO(LA := fbArbFullErr, FFO := ffo);
END_METHOD

// Test the BPTM seamlessly handles new requests at any stage
// Verify old requests are removed from arbiter
METHOD InterruptAtAllSteps
VAR_INPUT
END_VAR
VAR    
    //Final and transition assertions
    nTransitionID    :    UDINT := 16#DAAD;
    stTranReq    :    ST_BeamParams := PMPS_GVL.cst0RateBeam;
    
    nFirstReqID    :    UDINT    := 16#FEED;
    stFirstReq    :    ST_BeamParams := (nTran :=1, nRate := 16#FEED, neVRange :=2#1111_1111_1111_1111_1111_1111_1111_1111);
    
END_VAR
VAR_INST
    fbBPTM_InterruptionTest    :    BeamParameterTransitionManager;
    
    ffo : FB_HardwareFFOutput := (bAutoReset:=TRUE);
    fbSubSysIO : FB_DummyArbIO;
    fbBPR :  FB_BPRequestor;
    xFirstPass    :    BOOL := TRUE;
    eTestStep: E_BPTMTestStates := E_BPTMTestStates.Init;
    tonRetryTimeout : TON := (PT:=T#5s);
    
    fbBPTMDiscCycles : BeamParameterTransitionManager;
    fbSubSysIODisc : FB_DummyArbIO;
    fbArbDisc : FB_Arbiter(1000);
    
    iCount : UINT;
    
    aBPTM : ARRAY [1..cCycle] OF BeamParameterTransitionManager;
    BPTMUnderTest : REFERENCE TO BeamParameterTransitionManager;
    fbArbiter    :    FB_Arbiter(1);
    aArbIO : ARRAY [1..cCycle] OF FB_DummyArbIO;
    ArbIO : REFERENCE TO FB_DummyArbIO;
    nCycleLim : UINT;
    nCycle : UINT;
    sCurrentTestName : STRING :='';
    bCycleLimHit : BOOL; 
    nAllStepsDone : BYTE;
    tTimeOut : TON := (PT:=T#20ms);
        
    bTestedOnce : BOOl;
END_VAR
VAR CONSTANT
    nNewTarget : INT := 0;
    nRequestBP : INT := 1;
    nWaitForBP : INT := 2;
    nTransitioning : INT := 3;
    nWaitForFinalBP : INT := 4;
    nCleaningUp : INT := 5;
    nDone : INT := 6;
    nIdle : INT := 7;
END_VAR

(* These tests will confirm the BPTM is interruptable at any step,
meaning it will not deadlock or stall, and will always complete with
the correct sequencing *)

(* This functionality is crucial as a deadlocked BPTM will need manual intervention,
users of the BPTM should always be able to just set a target BP that is easy to reach
at any point in time, and have the BPTM head in that direction and succeed. *)

// Determine how many cycles it would take normally, to complete a full BPTM cycle
// This count will be verified against the current count constant

IF NOT bTestedOnce THEN

TEST('CheckBPTM Cycle Count');

WHILE fbBPTMDiscCycles.eBPTMState <> E_BPTMState.Idle DO
    
    fbBPTMDiscCycles.i_TransitionAssertionID := nTransitionID;
    fbBPTMDiscCycles.i_stTransitionAssertion := stTranReq;
    
    fbBPTMDiscCycles.i_nRequestedAssertionID := nFirstReqID;
    fbBPTMDiscCycles.i_stRequestedAssertion := stFirstReq;
    
    fbBPTMDiscCycles(fbArbiter:=fbArbDisc);
    fbSubSysIODisc(LA:=fbArbDisc, FFO:=ffo);
    
    fbBPTMDiscCycles.stCurrentBeamParameters := fbSubSysIODisc.q_stSimulatedBPReadback;
    
    fbSubSysIODisc.AutoUpdateBP := TRUE;
    
    fbBPTMDiscCycles.i_xDoneMoving S= fbBPTMDiscCycles.q_xTransitionAuthorized;
    
    iCount := iCount + 1;
END_WHILE

IF fbBPTMDiscCycles.eBPTMState = E_BPTMState.Idle THEN
    AssertTrue(cCycle >= iCount, CONCAT('cCycle is too low, increase it to', INT_TO_STRING(iCount)));
    TEST_FINISHED_NAMED('CheckBPTM Cycle Count');
END_IF

// Run BPTM for nCycleLim cycles, switch to a new target, verify BPTM completes anyways

FOR nCycleLim := 1 TO cCycle DO
    
    nCycle := 0;
    
    bCycleLimHit := FALSE;
    
    BPTMUnderTest REF= aBPTM[nCycleLim];
    ArbIO REF= aArbIO[nCycleLim];
    
    BPTMUnderTest.i_TransitionAssertionID := nTransitionID;
    BPTMUnderTest.i_stTransitionAssertion := stTranReq;
    
    ArbIO.AutoUpdateBP := TRUE;
    
    // Start the test for this Cycle Limit
    sCurrentTestName := CONCAT('CycleLimTest:',INT_TO_STRING(nCycleLim));
    TEST(sCurrentTestName);
    
    nAllStepsDone := 0;
    
    tTimeOut(IN:=FALSE);
        
    WHILE nAllStepsDone <> 16#FF DO
        
        tTimeOut(IN:= TRUE);

        IF tTimeOut.Q THEN
            AssertTrue(FALSE, CONCAT('Failed ', BYTE_TO_HEXSTR(nAllStepsDone, 2, FALSE)));
            EXIT;
        END_IF  
    
        // Verify all steps complete
        IF bCycleLimHit THEN
            nAllStepsDone.nNewTarget S= BPTMUnderTest.eBPTMState = E_BPTMState.NewTarget;
            nAllStepsDone.nRequestBP S= BPTMUnderTest.eBPTMState = E_BPTMState.RequestBP;
            nAllStepsDone.nWaitForBP S= BPTMUnderTest.eBPTMState = E_BPTMState.WaitForBP;
            nAllStepsDone.nTransitioning S= BPTMUnderTest.eBPTMState = E_BPTMState.Transitioning;
            nAllStepsDone.nWaitForFinalBP S= BPTMUnderTest.eBPTMState = E_BPTMState.WaitForFinalBP;
            nAllStepsDone.nCleaningUp S= BPTMUnderTest.eBPTMState = E_BPTMState.CleaningUp;
            nAllStepsDone.nDone S= BPTMUnderTest.eBPTMState = E_BPTMState.Done;
            nAllStepsDone.nIdle S= BPTMUnderTest.eBPTMState = E_BPTMState.Idle;
        ELSE
            nAllStepsDone := 0;
		END_IF
    
        // After nCycleLim cycles (nCycle), change the target
        IF nCycle >= nCycleLim THEN
            BPTMUnderTest.i_nRequestedAssertionID := nCycleLim;
            BPTMUnderTest.i_stRequestedAssertion.nRate := nCycleLim;
            bCycleLimHit := TRUE;
        ELSE
            BPTMUnderTest.i_nRequestedAssertionID := nFirstReqID;
            BPTMUnderTest.i_stRequestedAssertion := stFirstReq;
		END_IF
        
        BPTMUnderTest(fbArbiter:=fbArbiter);
        ArbIO(LA:=fbArbiter, FFO := ffo);
        
        BPTMUnderTest.stCurrentBeamParameters := ArbIO.q_stSimulatedBPReadback;
        
        BPTMUnderTest.i_xDoneMoving := BPTMUnderTest.q_xTransitionAuthorized;
        
        nCycle := nCycle + 1;
    
	END_WHILE
    
    AssertTrue(fbArbiter.CheckRequestInPool(BPTMUnderTest.i_nRequestedAssertionID),
        CONCAT('Final req not in pool: ', UINT_TO_STRING(nCycleLim)));
    AssertFalse(fbArbiter.CheckRequestInPool(BPTMUnderTest.i_TransitionAssertionID),
        'TransReq still in pool');
    AssertFalse(fbArbiter.CheckRequestInPool(nFirstReqID),
        'First req still in pool');
    AssertTrue(bCycleLimHit,
        CONCAT('Cycle lim not hit', UINT_TO_STRING(nCycleLim)));
    AssertTrue(ArbIO.q_stSimulatedBPReadback.nRate = BPTMUnderTest.i_stRequestedAssertion.nRate,
        'Rates are not equal...');
    
    TEST_FINISHED_NAMED(sCurrentTestName);
    
    // Clean up for next test
    
    fbArbiter.RemoveRequest(nFirstReqID);
    fbArbiter.RemoveRequest(nTransitionID);
    fbArbiter.RemoveRequest(nCycleLim);
    
END_FOR

END_IF
END_METHOD

END_FUNCTION_BLOCK

// TestComponents/FB_DiffBP_Test
{attribute 'call_after_init'}
FUNCTION_BLOCK FB_DiffBP_Test EXTENDS TcUnit.FB_TestSuite
VAR_INPUT
END_VAR
VAR_OUTPUT
END_VAR
VAR

END_VAR


BPDiff();

//Verify BP comparison remains logical.
METHOD BPDiff
VAR_INPUT
END_VAR
VAR
    BP1    :    ST_BeamParams;
    BP2    :    ST_BeamParams;
END_VAR
TEST('BPDiffCheck');

BP2.nTran := 10; 
    
AssertTrue(
    F_DifferentBeamParams(BP1, BP2),
    'DifferentBP eval is broken (True)'); 

BP1.nTran := BP2.nTran;   
    
AssertFalse(
    F_DifferentBeamParams(BP2, BP1),
    'DifferentBP eval is broken (False)');

TEST_FINISHED();
END_METHOD

END_FUNCTION_BLOCK

// TestComponents/FB_evRangeCalculator_Test
{attribute 'call_after_init'}
FUNCTION_BLOCK FB_evRangeCalculator_Test EXTENDS FB_TestSuite
VAR_INPUT
END_VAR
VAR_OUTPUT
END_VAR
VAR
END_VAR
VAR CONSTANT
    RandomBoundary : INT := 2;
END_VAR

BasicFunction();

METHOD BasicFunction
VAR_INPUT
END_VAR
VAR
    {attribute 'displaymode' := 'binary'}
    LastWord : DWORD := 2#0000_0000_0000_0000_0000_0000_0000_0010;
    {attribute 'displaymode' := 'binary'}
    Result : DWORD;
    {attribute 'displaymode' := 'binary'}
    TestEV : DWORD;
    
    {attribute 'displaymode' := 'binary'}
    tEvW : DWORD;
    tEv : REAL;
    
    
    fbStr : FB_FormatString;
    
    MiscNumber : INT;
END_VAR
VAR CONSTANT
    nLowerLimitBoundary : INT := 0;
    
    RandomBoundary : INT := 2;
    MNU : INT := 3; //RandomBoundary + 1
    MND : INT := 1; //RandomBoundary - 1
END_VAR
Test('CheckRanges');

//Lower limit equal
tEvW.nLowerLimitBoundary := TRUE;
tEv := PMPS_GVL.g_areVBoundaries[nLowerLimitBoundary];
Result := F_eVRangeCalculator(tEv, 0);
AssertTrue(
    Result = tEvW,
    'Lower limit not inclusive');
    
// Lower range flags
tEvW.nLowerLimitBoundary := TRUE;
tEv := PMPS_GVL.g_areVBoundaries[nLowerLimitBoundary] / 2;
Result := F_eVRangeCalculator(tEv, 0);
AssertTrue(
    Result = tEvW,
    'eV below lower range should come back true');
    
//Mid range
tEvW := 0;
tEvW.RandomBoundary := TRUE;
//ev result that is smack dab in the middle of a range
tEv := PMPS_GVL.g_areVBoundaries[RandomBoundary] - ((PMPS_GVL.g_areVBoundaries[RandomBoundary] - PMPS_GVL.g_areVBoundaries[MND]) / 2);
Result := F_eVRangeCalculator(tEv, 0);
AssertTrue(
    Result = tEvW,
    'In range failed, whatever you did, it broke this really bad.');

//Out of range
tEvW := 0;
tEvW.RandomBoundary := TRUE;
//Ev result that is beyond the current range (midway into the next range up)
tEv := PMPS_GVL.g_areVBoundaries[MNU] - (PMPS_GVL.g_areVBoundaries[MNU]-PMPS_GVL.g_areVBoundaries[RandomBoundary])/2;
Result := F_eVRangeCalculator(tEv, 0);
AssertFalse(
    Result = tEvW,
    'Out of range failed, whatever you did, it broke this really bad.');

TEST_FINISHED();

Test('Negative eV failsafes');
//Negative eV
AssertTrue(
    F_eVRangeCalculator(-300, 0) = 16#FFFF_FFFF,
    'Working with antimatter? Negative eV should failsafe to FFFF.');    

TEST_FINISHED();

Test('Out of range eV failsafes');
// eV too high
AssertTrue(
    F_eVRangeCalculator(PMPS_GVL.g_areVBoundaries[PMPS_GVL.g_cBoundaries] + 1, 0) = 16#FFFF_FFFF,
    'eV above the last threshold should failsafe.');    

TEST_FINISHED();

Test('Check hyst keeps');

LastWord := F_eVRangeCalculator(PMPS_GVL.g_areVBoundaries[RandomBoundary], 2#0000_0000_0000_0000_0000_0000_0000_0000);

// Last word should be 2#0000_0000_0000_0100

    Result := F_eVRangeCalculator(
        PMPS_GVL.g_areVBoundaries[RandomBoundary] + PMPS_GVL.reVHyst - PMPS_GVL.reVHyst/2,
         LastWord);
    TestEV := 0;
    TestEV.RandomBoundary := TRUE;
    TestEV.MNU := True;
 
    fbStr.arg1 := F_DWORD(Result);
    fbStr.arg2 := F_DWORD(TestEV);
    fbStr.sFormat := 'Moving up does not stick. Result: %b vs. Test: %b';
    fbStr();
        
AssertTrue(Result = TestEV,
    fbStr.sOut);
    
    Result := F_eVRangeCalculator(
        PMPS_GVL.g_areVBoundaries[RandomBoundary - 1] - PMPS_GVL.reVHyst + PMPS_GVL.reVHyst/2, 
        LastWord);
    TestEV := 0;
    TestEV.RandomBoundary := TRUE;
    TestEV.MND := True;
    
    fbStr.arg1 := F_DWORD(Result);
    fbStr.arg2 := F_DWORD(TestEV);
    fbStr.sFormat := 'Moving down does not stick. Result: %b vs. Test: %b';
    fbStr();
    
AssertTrue(Result = TestEV,
    fbStr.sOut);

TEST_FINISHED();

Test('Check hyst drops');

    Result := F_eVRangeCalculator(
        PMPS_GVL.g_areVBoundaries[MND] - PMPS_GVL.reVHyst*1.1, 
        LastWord);
    TestEV := 0;
    TestEV.MND := TRUE;
    
    fbStr.arg1 := F_DWORD(Result);
    fbStr.arg2 := F_DWORD(TestEV);
    fbStr.sFormat := 'Moving down does not drop. Result: %b vs. Test: %b';
    fbStr();
    
AssertTrue(Result = TestEV,
    fbStr.sOut);

    Result := F_eVRangeCalculator(
        PMPS_GVL.g_areVBoundaries[RandomBoundary] + PMPS_GVL.reVHyst*1.1, 
        LastWord);
    TestEV := 0;
    TestEV.MNU := TRUE;
    
    fbStr.arg1 := F_DWORD(Result);
    fbStr.arg2 := F_DWORD(TestEV);
    fbStr.sFormat := 'Moving up does not drop. Result: %b vs. Test: %b';
    fbStr();
    
AssertTrue(Result = TestEV,
    fbStr.sOut);

TEST_FINISHED();
END_METHOD

END_FUNCTION_BLOCK

// TestComponents/FB_eVWithinSpec_Test
{attribute 'call_after_init'}
FUNCTION_BLOCK FB_eVWithinSpec_Test EXTENDS TcUnit.FB_TestSuite
VAR_INPUT
END_VAR
VAR_OUTPUT
END_VAR
VAR
END_VAR

evWithinRangeChecks();

METHOD evWithinRangeChecks
VAR_INPUT
END_VAR
VAR

END_VAR
TEST('evWithinRangeChecks');
    
//Upper limit equal
AssertTrue(
    F_eVWithinSpec(300, 2#0000_0000_0000_0010),
    'Upper limit not inclusive');
//Lower limit equal
AssertTrue(
    F_eVWithinSpec(300, 2#0000_0000_0000_0100),
    'Lower limit not inclusive');
//Out of range
AssertFalse(
    F_eVWithinSpec(300.1, 2#0000_0000_0000_0010),
    'Out of range failed, whatever you did, it broke this really bad.');
//Negative eV
AssertFalse(
    F_eVWithinSpec(-300, 16#FFFF),
    'Working with antimatter? Negative eV should not be acceptable.');
//Upper unallocated range
AssertFalse(
    F_eVWithinSpec(1701, 2#1000_0000_0000_0000),
    'eV range should not evaluate past 1.7keV');
    
TEST_FINISHED();
END_METHOD

END_FUNCTION_BLOCK

// TestComponents/FB_FastFault_Test
{attribute 'call_after_init'}
FUNCTION_BLOCK FB_FastFault_Test EXTENDS TcUnit.FB_TestSuite
VAR_INPUT
END_VAR
VAR_OUTPUT
END_VAR
VAR
	fbTime : FB_LocalSystemTime := ( bEnable := TRUE, dwCycle := 1 ); //Get current system time, used for override
END_VAR
VAR CONSTANT
    OvrdTime : TIME := T#2s;
END_VAR

FFCombinedFunctionality();
FFRegistration();
FFOvrdAndNextFault();

METHOD FFCombinedFunctionality
VAR_INPUT
END_VAR
VAR_INST
    fbFF    :    FB_FastFault;
    fbFFO    :    FB_HardwareFFOutput;
    
END_VAR
TEST('FFCombinedFunctionality');

//Clear initial faults
fbFFO.i_xReset:=TRUE; //Reset requested at start of cycle

fbFF(io_fbFFHWO := fbFFO, //FF reset somehwere in code
    i_xOK := TRUE,
    i_xReset := TRUE);

fbFFO.EvaluateOutput(); //FFO eval called at end of cycle
    
AssertTrue(fbFFO.q_xFastFaultOut,
    'Fast fault did not clear');


//Induce fault with FF

fbFFO(i_xReset := FALSE); //Reset released at start of cycle

fbFF(io_fbFFHWO := fbFFO, //FF faulted
    i_xOK := FALSE); //Reset is still set true from last call.
    
fbFFO.EvaluateOutput(); //FFO eval called at end of cycle

AssertFalse(fbFFO.q_xFastFaultOut,
    'Fast fault did not trip the beam');
    
    
//FFO remains faulted until local (FF) and FFO receieve fresh reset request, and faults
//are actually cleared

//Attempt to clear FFO fails because FF still faulted
fbFFO.i_xReset := TRUE; //Reset requested

fbFF(io_fbFFHWO := fbFFO, //FF faulted
    i_xOK := FALSE,
    i_xReset := FALSE);
    
fbFFO.EvaluateOutput(); //FFO eval called at end of cycle

AssertFalse(fbFFO.q_xFastFaultOut,
    'Fast fault output cleared while fault remains, very bad');
    
//Attempt to clear FF while fault remains fails
fbFFO.EvaluateOutput(i_xReset := FALSE);

fbFFO.i_xReset := TRUE; //Reset requested

fbFF(io_fbFFHWO := fbFFO, //FF faulted
    i_xOK := FALSE,
    i_xReset := TRUE); //This reset should fail.
    
fbFFO.EvaluateOutput(); //FFO eval called at end of cycle

AssertFalse(fbFFO.q_xFastFaultOut,
    'Fast fault cleared while fault remains, very bad');
    
TEST_FINISHED();
END_METHOD

METHOD FFOvrdAndNextFault
VAR_INPUT
END_VAR
VAR_INST
    fbFF    :    FB_FastFault :=(
        i_xAutoReset := TRUE);
    fbFFO    :    FB_HardwareFFOutput := (i_sNetID:='',
        bAutoReset := TRUE);
    rFF : REFERENCE TO ST_FF;
    
    FirstPass : BOOL := TRUE;
	fbTimePass : BOOL := TRUE;
    OvrdActvTstDone : BOOL := FALSE;
    
    TestsDone : BOOL := FALSE;
	Now: DATE_AND_TIME;
	Expiration : DINT; 
	OvdTime : TIME ;
	Expire: TIMESTRUCT;
//seconds:ULINT;
	specificLocalTimeToFileTime : FB_TzSpecificLocalTimeToFileTime;
    fileTime: T_FILETIME;
END_VAR
TEST('FFVetoAndNextFault');
fbTime();

// I noticed something weird going on with the PEWatcher on the L line. It was faulted, and the fast fault
// was not tripping off beam. It had been previously overridden so I was wondering why it wasn't causing a trip.

IF  FirstPass  THEN

    fbFF(io_fbFFHWO := fbFFO, //FF reset somehwere in code
        i_xOK := TRUE);
    
    fbFFO.ExecuteNoLog(); //FFO eval called at end of cycle
        
    AssertTrue(fbFFO.q_xFastFaultOut,
        'Fast fault did not clear');
    
    
    //Induce fault with FF
    
    fbFF(io_fbFFHWO := fbFFO, //FF faulted
        i_xOK := FALSE); 
        
    fbFFO.ExecuteNoLog(); //FFO eval called at end of cycle
    
    AssertFalse(fbFFO.q_xFastFaultOut,
        'Fast fault did not trip the beam');

    rFF REF= fbFFO.astFF[fbFF.RegistrationIdx];
	
FirstPass := FALSE; 
    
END_IF


IF fbTime.bValid AND fbTimePass  THEN
	
	Now := SystemTime_TO_DT(fbTime.systemTime);
	Expire:= fbTime.systemTime;
	Expire.wSecond:= Expire.wSecond+5;
	specificLocalTimeToFileTime(in := Tc2_Utilities.SYSTEMTIME_TO_FILETIME(Expire), tzInfo := , out => fileTime);
	Expiration := TO_DINT((SHL(DWORD_TO_ULINT(fileTime.dwHighDateTime), 32) + DWORD_TO_ULINT(fileTime.dwLowDateTime)) / 10000000 - 11644473600);;

    WRITE_PROTECTED_DINT(ADR(rFF.Ovrd.Expiration), Expiration );
	WRITE_PROTECTED_TIME(ADR(rFF.Ovrd.Timer.PT), OvrdTime );
    WRITE_PROTECTED_BOOL(ADR(rFF.Ovrd.Activate), TRUE);
	
	fbTimePass:=FALSE;
    
END_IF

// On every cycle:
fbFF(io_fbFFHWO := fbFFO, //FF faulted
    i_xOK := FALSE); 
    
fbFFO.ExecuteNoLog(); //FFO eval called at end of cycle


IF rFF.Ovrd.Active AND rFF.BeamPermitted THEN

    AssertTrue(fbFFO.q_xFastFaultOut,
        'Fast fault should be overridden so FFO should be true');
    
    OvrdActvTstDone := TRUE;
END_IF

IF OvrdActvTstDone and NOT rFF.Ovrd.Active and not rff.BeamPermitted THEN
    
    AssertFalse(fbFFO.q_xFastFaultOut,
        'Fast fault override expired so beam should be off.');
   // AssertFalse(rFF.BeamPermitted, 'Beam should not be permitted now');
    
    TestsDone := TRUE;
END_IF


IF TestsDone THEN    
    TEST_FINISHED_NAMED('FFVetoAndNextFault');
END_IF
END_METHOD

METHOD FFRegistration
VAR_INPUT
END_VAR
VAR_INST
    fbFF    :    FB_FastFault;
    fbFFO    :    FB_HardwareFFOutput;
    astFF : ARRAY[0..10] OF ST_FF;
END_VAR
TEST('FFRegistration');

fbFF(io_fbFFHWO := fbFFO);

AssertEquals_STRING(fbFF.sPath, fbFFO.astFF[fbFF.RegistrationIdx].Info.sPath,
    'FF registration with FFO did not succeed');

TEST_FINISHED();
END_METHOD

END_FUNCTION_BLOCK

// TestComponents/FB_PhotonEnergyWatcher_Test
{attribute 'call_after_init'}
FUNCTION_BLOCK FB_PhotonEnergyWatcher_Test EXTENDS TcUnit.FB_TestSuite
VAR_INPUT
END_VAR
VAR_OUTPUT
END_VAR
VAR

END_VAR

PEWatcherBasicFunction();

METHOD PEWatcherBasicFunction
VAR_INPUT
END_VAR
VAR_INST
    fbPEW    :    FB_PhotonEnergyWatcher;
    fbFFO    :    FB_HardwareFFOutput;
    q_Output    :    BOOL;
    
